C05454=1045.852,-21.922,423.875,169.880,34.118,156.433
C05455=1045.858,-21.672,423.861,169.882,34.118,156.433
C05456=1045.864,-21.423,423.847,169.883,34.120,156.434
C05457=1045.870,-21.174,423.834,169.885,34.121,156.434
C05458=1045.877,-20.923,423.819,169.887,34.122,156.434
C05459=1045.883,-20.675,423.805,169.889,34.124,156.434
C05460=1045.890,-20.425,423.792,169.891,34.125,156.434
C05461=1045.895,-20.175,423.778,169.893,34.126,156.434
C05462=1045.902,-19.925,423.764,169.895,34.127,156.435
C05463=1045.908,-19.676,423.750,169.897,34.129,156.435
C05464=1045.916,-19.394,423.734,169.899,34.130,156.435
C05465=1045.922,-19.113,423.719,169.901,34.131,156.435
C05466=1045.930,-18.831,423.702,169.904,34.133,156.435
C05467=1045.937,-18.550,423.687,169.906,34.134,156.436
C05468=1045.943,-18.300,423.673,169.908,34.136,156.436
C05469=1045.949,-18.051,423.658,169.910,34.137,156.436
C05470=1045.956,-17.801,423.645,169.912,34.138,156.436
C05471=1045.962,-17.552,423.632,169.914,34.140,156.436
C05472=1045.969,-17.302,423.617,169.915,34.141,156.436
C05473=1045.975,-17.053,423.603,169.917,34.142,156.437
C05474=1045.981,-16.803,423.588,169.919,34.143,156.437
C05475=1045.987,-16.554,423.575,169.921,34.145,156.437
C05476=1045.993,-16.303,423.561,169.923,34.146,156.437
C05477=1046.001,-16.054,423.547,169.925,34.147,156.437
C05478=1046.007,-15.805,423.533,169.927,34.148,156.438
C05479=1046.013,-15.555,423.518,169.929,34.150,156.438
C05480=1046.019,-15.306,423.505,169.931,34.151,156.438
C05481=1046.026,-15.056,423.490,169.933,34.152,156.438
C05482=1046.031,-14.807,423.476,169.935,34.154,156.438
C05483=1046.038,-14.557,423.462,169.938,34.155,156.439
C05484=1046.044,-14.308,423.448,169.940,34.157,156.439
C05485=1046.050,-14.058,423.433,169.941,34.158,156.439
C05486=1046.057,-13.808,423.419,169.943,34.159,156.439
C05487=1046.063,-13.559,423.405,169.945,34.161,156.439
C05488=1046.069,-13.309,423.391,169.947,34.162,156.440
C05489=1046.075,-13.060,423.377,169.949,34.163,156.440
C05490=1046.082,-12.810,423.362,169.951,34.165,156.440
C05491=1046.087,-12.561,423.348,169.953,34.166,156.440
C05492=1046.094,-12.312,423.333,169.955,34.168,156.440
C05493=1046.100,-12.062,423.320,169.957,34.169,156.441
C05494=1046.106,-11.812,423.305,169.958,34.170,156.441
C05495=1046.113,-11.562,423.291,169.960,34.172,156.441
C05496=1046.119,-11.314,423.276,169.962,34.173,156.441
C05497=1046.125,-11.064,423.262,169.964,34.174,156.441
C05498=1046.131,-10.815,423.248,169.966,34.176,156.442
C05499=1046.138,-10.565,423.233,169.968,34.177,156.442
C05500=1046.144,-10.315,423.218,169.970,34.178,156.442
C05501=1046.150,-10.066,423.205,169.972,34.180,156.442
C05502=1046.157,-9.816,423.190,169.974,34.181,156.442
C05503=1046.163,-9.567,423.175,169.975,34.183,156.443
C05504=1046.169,-9.317,423.161,169.977,34.184,156.443
C05505=1046.176,-9.068,423.147,169.979,34.185,156.443
C05506=1046.182,-8.818,423.132,169.981,34.187,156.443
C05507=1046.188,-8.569,423.118,169.983,34.188,156.443
C05508=1046.195,-8.319,423.104,169.985,34.189,156.444
C05509=1046.201,-8.070,423.089,169.987,34.191,156.444
C05510=1046.207,-7.821,423.074,169.989,34.192,156.444
C05511=1046.213,-7.570,423.060,169.990,34.194,156.444
C05512=1046.220,-7.321,423.046,169.992,34.195,156.444
C05513=1046.226,-7.072,423.031,169.994,34.196,156.445
C05514=1046.232,-6.822,423.016,169.996,34.198,156.445
C05515=1046.239,-6.572,423.003,169.998,34.199,156.445
C05516=1046.245,-6.323,422.988,170.001,34.200,156.445
C05517=1046.251,-6.074,422.973,170.003,34.202,156.445
C05518=1046.258,-5.824,422.958,170.005,34.203,156.446
C05519=1046.264,-5.575,422.945,170.006,34.205,156.446
C05520=1046.270,-5.325,422.930,170.008,34.206,156.446
C05521=1046.277,-5.076,422.915,170.010,34.207,156.446
C05522=1046.283,-4.826,422.900,170.012,34.209,156.446
C05523=1046.290,-4.577,422.886,170.014,34.210,156.447
C05524=1046.296,-4.328,422.871,170.016,34.211,156.447
C05525=1046.302,-4.077,422.857,170.018,34.213,156.447
C05526=1046.308,-3.828,422.842,170.019,34.214,156.447
C05527=1046.315,-3.579,422.828,170.021,34.215,156.447
C05528=1046.322,-3.296,422.811,170.023,34.217,156.448
C05529=1046.329,-3.012,422.794,170.025,34.219,156.448
C05530=1046.336,-2.729,422.778,170.028,34.220,156.448
C05531=1046.343,-2.446,422.760,170.030,34.222,156.448
C05532=1046.350,-2.196,422.745,170.031,34.224,156.449
C05533=1046.355,-1.947,422.731,170.033,34.225,156.449
C05534=1046.362,-1.698,422.716,170.035,34.226,156.449
C05535=1046.368,-1.448,422.701,170.037,34.228,156.449
C05536=1046.374,-1.199,422.686,170.039,34.230,156.450
C05537=1046.380,-0.950,422.671,170.041,34.231,156.450
C05538=1046.387,-0.700,422.657,170.042,34.232,156.450
C05539=1046.393,-0.450,422.642,170.044,34.234,156.450
C05540=1046.399,-0.201,422.627,170.046,34.236,156.450
C05541=1046.404,0.049,422.611,170.048,34.237,156.451
C05542=1046.411,0.298,422.597,170.050,34.239,156.451
C05543=1046.417,0.548,422.582,170.052,34.240,156.451
C05544=1046.423,0.797,422.567,170.054,34.241,156.451
C05545=1046.429,1.047,422.552,170.056,34.243,156.452
C05546=1046.436,1.296,422.537,170.058,34.245,156.452
C05547=1046.442,1.546,422.522,170.060,34.246,156.452
C05548=1046.448,1.795,422.508,170.062,34.247,156.452
C05549=1046.454,2.045,422.493,170.063,34.249,156.452
C05550=1046.461,2.294,422.478,170.065,34.250,156.453
C05551=1046.467,2.544,422.463,170.067,34.252,156.453
C05552=1046.474,2.793,422.447,170.069,34.253,156.453
C05553=1046.480,3.042,422.433,170.071,34.255,156.453
C05554=1046.486,3.292,422.418,170.072,34.256,156.454
C05555=1046.492,3.541,422.403,170.074,34.257,156.454
C05556=1046.498,3.791,422.387,170.076,34.259,156.454
C05557=1046.504,4.041,422.372,170.078,34.261,156.454
C05558=1046.511,4.290,422.357,170.080,34.262,156.454
C05559=1046.517,4.539,422.342,170.081,34.264,156.455
C05560=1046.523,4.788,422.327,170.083,34.265,156.455
C05561=1046.530,5.038,422.312,170.085,34.267,156.455
C05562=1046.536,5.288,422.297,170.087,34.268,156.455
C05563=1046.542,5.537,422.282,170.089,34.270,156.456
C05564=1046.549,5.787,422.267,170.090,34.271,156.456
C05565=1046.555,6.035,422.252,170.092,34.272,156.456
C05566=1046.561,6.285,422.237,170.094,34.274,156.456
C05567=1046.567,6.535,422.221,170.097,34.276,156.457
C05568=1046.573,6.785,422.206,170.099,34.277,156.457
C05569=1046.580,7.034,422.191,170.100,34.278,156.457
C05570=1046.586,7.283,422.176,170.102,34.280,156.457
C05571=1046.593,7.533,422.161,170.104,34.282,156.457
C05572=1046.599,7.783,422.146,170.106,34.283,156.458
C05573=1046.606,8.032,422.130,170.108,34.284,156.458
C05574=1046.612,8.281,422.116,170.109,34.286,156.458
C05575=1046.617,8.531,422.100,170.111,34.287,156.458
C05576=1046.624,8.780,422.085,170.113,34.289,156.459
C05577=1046.630,9.029,422.070,170.115,34.291,156.459
C05578=1046.637,9.279,422.055,170.117,34.292,156.459
C05579=1046.643,9.529,422.040,170.118,34.293,156.459
C05580=1046.650,9.778,422.024,170.120,34.295,156.459
C05581=1046.656,10.027,422.009,170.122,34.297,156.460
C05582=1046.662,10.277,421.994,170.124,34.298,156.460
C05583=1046.668,10.526,421.978,170.126,34.299,156.460
C05584=1046.675,10.776,421.963,170.127,34.301,156.460
C05585=1046.681,11.026,421.948,170.129,34.302,156.461
C05586=1046.688,11.275,421.932,170.131,34.304,156.461
C05587=1046.694,11.524,421.917,170.133,34.305,156.461
C05588=1046.701,11.774,421.902,170.135,34.307,156.461
C05589=1046.707,12.023,421.887,170.136,34.308,156.461
C05590=1046.713,12.273,421.871,170.139,34.309,156.462
C05591=1046.720,12.522,421.856,170.141,34.311,156.462
C05592=1046.727,12.807,421.838,170.143,34.313,156.462
C05593=1046.734,13.092,421.821,170.145,34.315,156.463
C05594=1046.741,13.378,421.804,170.147,34.316,156.463
C05595=1046.749,13.663,421.786,170.149,34.318,156.463
C05596=1046.756,13.912,421.770,170.151,34.319,156.463
C05597=1046.762,14.162,421.755,170.153,34.321,156.463
C05598=1046.768,14.411,421.739,170.154,34.322,156.464
C05599=1046.774,14.661,421.724,170.156,34.324,156.464
C05600=1046.781,14.910,421.708,170.158,34.325,156.464
C05601=1046.787,15.160,421.693,170.160,34.327,156.464
C05602=1046.793,15.409,421.677,170.161,34.329,156.465
C05603=1046.799,15.659,421.662,170.163,34.330,156.465
C05604=1046.806,15.908,421.646,170.165,34.332,156.465
C05605=1046.812,16.157,421.631,170.167,34.333,156.465
C05606=1046.818,16.407,421.615,170.168,34.335,156.466
C05607=1046.825,16.656,421.599,170.170,34.336,156.466
C05608=1046.830,16.906,421.584,170.172,34.338,156.466
C05609=1046.837,17.155,421.568,170.174,34.340,156.466
C05610=1046.843,17.404,421.553,170.175,34.341,156.467
C05611=1046.849,17.654,421.537,170.178,34.343,156.467
C05612=1046.856,17.903,421.522,170.180,34.344,156.467
C05613=1046.862,18.153,421.506,170.182,34.346,156.467
C05614=1046.868,18.402,421.490,170.183,34.347,156.468
C05615=1046.875,18.651,421.475,170.185,34.349,156.468
C05616=1046.881,18.901,421.459,170.187,34.350,156.468
C05617=1046.887,19.150,421.443,170.189,34.352,156.468
C05618=1046.893,19.400,421.427,170.190,34.353,156.469
C05619=1046.900,19.649,421.412,170.192,34.355,156.469
C05620=1046.906,19.898,421.396,170.194,34.357,156.469
C05621=1046.912,20.148,421.381,170.196,34.358,156.469
C05622=1046.918,20.397,421.364,170.197,34.360,156.470
C05623=1046.925,20.646,421.349,170.199,34.362,156.470
C05624=1046.930,20.896,421.333,170.201,34.363,156.470
C05625=1046.937,21.145,421.317,170.203,34.365,156.470
C05626=1046.943,21.394,421.301,170.204,34.366,156.471
C05627=1046.950,21.644,421.285,170.206,34.368,156.471
C05628=1046.956,21.894,421.270,170.208,34.370,156.471
C05629=1046.963,22.143,421.254,170.209,34.371,156.471
C05630=1046.969,22.393,421.238,170.212,34.373,156.472
C05631=1046.975,22.642,421.222,170.214,34.374,156.472
C05632=1046.981,22.892,421.207,170.216,34.376,156.472
C05633=1046.987,23.141,421.190,170.217,34.377,156.472
C05634=1046.994,23.390,421.175,170.219,34.379,156.473
C05635=1046.999,23.639,421.158,170.221,34.381,156.473
C05636=1047.006,23.888,421.143,170.223,34.382,156.473
C05637=1047.012,24.139,421.127,170.224,34.383,156.473
C05638=1047.019,24.388,421.111,170.226,34.385,156.474
C05639=1047.025,24.637,421.095,170.228,34.387,156.474
C05640=1047.031,24.887,421.079,170.229,34.388,156.474
C05641=1047.038,25.136,421.063,170.231,34.390,156.474
C05642=1047.044,25.385,421.047,170.233,34.391,156.475
C05643=1047.050,25.635,421.032,170.235,34.393,156.475
C05644=1047.057,25.885,421.015,170.236,34.395,156.475
C05645=1047.063,26.134,420.999,170.238,34.396,156.475
C05646=1047.069,26.383,420.983,170.240,34.398,156.476
C05647=1047.075,26.633,420.967,170.241,34.399,156.476
C05648=1047.082,26.882,420.951,170.244,34.401,156.476
C05649=1047.088,27.131,420.935,170.246,34.403,156.476
C05650=1047.094,27.381,420.918,170.248,34.404,156.477
C05651=1047.101,27.630,420.903,170.249,34.406,156.477
C05652=1047.107,27.879,420.887,170.251,34.407,156.477
C05653=1047.113,28.129,420.870,170.253,34.409,156.477
C05654=1047.119,28.378,420.855,170.254,34.411,156.478
C05655=1047.125,28.628,420.839,170.256,34.413,156.478
C05656=1047.133,28.914,420.820,170.258,34.414,156.478
C05657=1047.140,29.200,420.802,170.260,34.416,156.479
C05658=1047.147,29.486,420.783,170.262,34.418,156.479
C05659=1047.154,29.773,420.764,170.264,34.420,156.479
C05660=1047.160,30.022,420.748,170.266,34.421,156.479
C05661=1047.167,30.271,420.732,170.267,34.423,156.480
C05662=1047.173,30.521,420.715,170.269,34.425,156.480
C05663=1047.179,30.771,420.699,170.271,34.427,156.480
C05664=1047.185,31.020,420.683,170.272,34.428,156.480
C05665=1047.191,31.270,420.667,170.275,34.430,156.481
C05666=1047.198,31.519,420.651,170.277,34.431,156.481
C05667=1047.204,31.769,420.634,170.279,34.433,156.481
C05668=1047.210,32.018,420.618,170.280,34.434,156.481
C05669=1047.216,32.267,420.602,170.282,34.436,156.482
C05670=1047.222,32.517,420.586,170.284,34.438,156.482
C05671=1047.230,32.766,420.569,170.285,34.440,156.482
C05672=1047.236,33.015,420.553,170.287,34.441,156.483
C05673=1047.242,33.264,420.536,170.289,34.443,156.483
C05674=1047.248,33.514,420.520,170.290,34.444,156.483
C05675=1047.254,33.764,420.503,170.292,34.446,156.483
C05676=1047.261,34.013,420.488,170.294,34.448,156.484
C05677=1047.267,34.262,420.471,170.295,34.450,156.484
C05678=1047.273,34.512,420.455,170.297,34.451,156.484
C05679=1047.280,34.761,420.438,170.299,34.453,156.484
C05680=1047.286,35.010,420.422,170.301,34.454,156.485
C05681=1047.292,35.260,420.405,170.303,34.456,156.485
C05682=1047.298,35.509,420.390,170.305,34.458,156.485
C05683=1047.305,35.759,420.373,170.307,34.460,156.486
C05684=1047.311,36.008,420.356,170.308,34.461,156.486
C05685=1047.317,36.257,420.340,170.310,34.462,156.486
C05686=1047.324,36.507,420.323,170.312,34.464,156.486
C05687=1047.330,36.756,420.307,170.313,34.465,156.487
C05688=1047.336,37.006,420.291,170.315,34.467,156.487
C05689=1047.343,37.255,420.274,170.317,34.469,156.487
C05690=1047.349,37.504,420.258,170.318,34.471,156.487
C05691=1047.355,37.753,420.241,170.320,34.472,156.488
C05692=1047.362,38.003,420.224,170.322,34.474,156.488
C05693=1047.368,38.252,420.208,170.323,34.476,156.488
C05694=1047.374,38.502,420.192,170.325,34.477,156.488
C05695=1047.380,38.751,420.175,170.327,34.479,156.489
C05696=1047.387,39.000,420.158,170.328,34.481,156.489
C05697=1047.393,39.250,420.142,170.331,34.483,156.489
C05698=1047.398,39.499,420.124,170.333,34.484,156.490
C05699=1047.405,39.749,420.108,170.334,34.486,156.490
C05700=1047.411,39.998,420.091,170.336,34.488,156.490
C05701=1047.417,40.247,420.074,170.338,34.489,156.490
C05702=1047.423,40.497,420.058,170.339,34.491,156.491
C05703=1047.429,40.746,420.041,170.341,34.492,156.491
C05704=1047.436,40.995,420.024,170.343,34.494,156.491
C05705=1047.442,41.245,420.008,170.344,34.496,156.491
C05706=1047.448,41.494,419.991,170.346,34.498,156.492
C05707=1047.454,41.743,419.975,170.348,34.500,156.492
C05708=1047.461,41.993,419.958,170.349,34.501,156.492
C05709=1047.467,42.242,419.941,170.351,34.503,156.493
C05710=1047.473,42.491,419.925,170.353,34.504,156.493
C05711=1047.480,42.741,419.907,170.355,34.506,156.493
C05712=1047.486,42.990,419.891,170.357,34.508,156.493
C05713=1047.491,43.239,419.874,170.359,34.510,156.494
C05714=1047.498,43.489,419.857,170.360,34.511,156.494
C05715=1047.504,43.738,419.840,170.362,34.513,156.494
C05716=1047.511,43.988,419.823,170.364,34.515,156.495
C05717=1047.516,44.237,419.806,170.365,34.517,156.495
C05718=1047.522,44.486,419.790,170.367,34.518,156.495
C05719=1047.529,44.736,419.772,170.369,34.520,156.495
C05720=1047.536,45.022,419.753,170.371,34.522,156.496
C05721=1047.543,45.308,419.733,170.372,34.524,156.496
C05722=1047.549,45.595,419.714,170.374,34.526,156.496
C05723=1047.557,45.881,419.695,170.376,34.528,156.497
C05724=1047.562,46.130,419.678,170.378,34.530,156.497
C05725=1047.569,46.380,419.660,170.380,34.532,156.497
C05726=1047.575,46.629,419.644,170.382,34.533,156.498
C05727=1047.581,46.879,419.626,170.384,34.535,156.498
C05728=1047.587,47.128,419.610,170.385,34.537,156.498
C05729=1047.593,47.377,419.593,170.387,34.538,156.498
C05730=1047.600,47.626,419.575,170.389,34.540,156.499
C05731=1047.606,47.876,419.559,170.390,34.542,156.499
C05732=1047.612,48.125,419.541,170.392,34.544,156.499
C05733=1047.618,48.374,419.524,170.394,34.545,156.500
C05734=1047.624,48.624,419.507,170.395,34.547,156.500
C05735=1047.631,48.873,419.490,170.397,34.549,156.500
C05736=1047.636,49.122,419.473,170.398,34.551,156.501
C05737=1047.643,49.372,419.456,170.400,34.553,156.501
C05738=1047.649,49.621,419.439,170.402,34.554,156.501
C05739=1047.655,49.871,419.421,170.404,34.556,156.501
C05740=1047.661,50.120,419.405,170.406,34.558,156.502
C05741=1047.667,50.369,419.388,170.408,34.559,156.502
C05742=1047.673,50.618,419.370,170.409,34.561,156.502
C05743=1047.679,50.868,419.354,170.411,34.563,156.503
C05744=1047.686,51.117,419.336,170.413,34.564,156.503
C05745=1047.692,51.366,419.319,170.414,34.566,156.503
C05746=1047.699,51.616,419.301,170.416,34.568,156.503
C05747=1047.704,51.865,419.285,170.418,34.570,156.504
C05748=1047.711,52.115,419.267,170.419,34.572,156.504
C05749=1047.717,52.363,419.250,170.421,34.574,156.504
C05750=1047.723,52.613,419.232,170.422,34.575,156.505
C05751=1047.729,52.862,419.215,170.424,34.577,156.505
C05752=1047.736,53.112,419.199,170.427,34.579,156.505
C05753=1047.741,53.361,419.181,170.428,34.580,156.505
C05754=1047.748,53.610,419.164,170.430,34.582,156.506
C05755=1047.754,53.859,419.146,170.432,34.583,156.506
C05756=1047.761,54.109,419.129,170.433,34.585,156.506
C05757=1047.767,54.358,419.113,170.435,34.587,156.507
C05758=1047.773,54.608,419.095,170.437,34.589,156.507
C05759=1047.779,54.857,419.078,170.438,34.590,156.507
C05760=1047.786,55.106,419.060,170.440,34.592,156.507
C05761=1047.792,55.356,419.042,170.442,34.594,156.508
C05762=1047.798,55.605,419.025,170.443,34.596,156.508
C05763=1047.804,55.854,419.008,170.445,34.598,156.508
C05764=1047.810,56.104,418.991,170.446,34.599,156.509
C05765=1047.817,56.353,418.974,170.449,34.601,156.509
C05766=1047.823,56.602,418.956,170.451,34.602,156.509
C05767=1047.830,56.852,418.939,170.452,34.604,156.509
C05768=1047.835,57.101,418.921,170.454,34.606,156.510
C05769=1047.842,57.350,418.904,170.456,34.607,156.510
C05770=1047.849,57.600,418.887,170.457,34.609,156.510
C05771=1047.854,57.849,418.869,170.459,34.611,156.511
C05772=1047.861,58.098,418.852,170.461,34.613,156.511
C05773=1047.867,58.347,418.834,170.462,34.615,156.511
C05774=1047.874,58.596,418.817,170.464,34.616,156.511
C05775=1047.880,58.846,418.800,170.466,34.618,156.512
C05776=1047.886,59.095,418.782,170.467,34.620,156.512
C05777=1047.893,59.344,418.765,170.469,34.621,156.512
C05778=1047.899,59.595,418.748,170.472,34.623,156.513
C05779=1047.905,59.843,418.731,170.473,34.624,156.513
C05780=1047.911,60.093,418.713,170.475,34.626,156.513
C05781=1047.917,60.342,418.696,170.476,34.628,156.513
C05782=1047.924,60.591,418.678,170.478,34.630,156.514
C05783=1047.931,60.840,418.660,170.480,34.632,156.514
C05784=1047.937,61.126,418.640,170.482,34.634,156.514
C05785=1047.944,61.412,418.620,170.484,34.635,156.515
C05786=1047.953,61.699,418.600,170.485,34.637,156.515
C05787=1047.960,61.985,418.580,170.487,34.639,156.515
C05788=1047.966,62.234,418.562,170.489,34.641,156.516
C05789=1047.972,62.483,418.545,170.491,34.643,156.516
C05790=1047.978,62.733,418.527,170.493,34.645,156.516
C05791=1047.985,62.982,418.510,170.495,34.646,156.516
C05792=1047.991,63.231,418.492,170.497,34.648,156.517
C05793=1047.998,63.480,418.474,170.498,34.649,156.517
C05794=1048.005,63.730,418.457,170.500,34.651,156.517
C05795=1048.010,63.979,418.439,170.502,34.652,156.517
C05796=1048.016,64.228,418.421,170.503,34.654,156.518
C05797=1048.023,64.478,418.404,170.505,34.656,156.518
C05798=1048.029,64.727,418.386,170.506,34.658,156.518
C05799=1048.035,64.977,418.369,170.508,34.660,156.519
C05800=1048.042,65.225,418.351,170.510,34.661,156.519
C05801=1048.048,65.475,418.333,170.511,34.663,156.519
C05802=1048.054,65.724,418.315,170.513,34.665,156.520
C05803=1048.060,65.974,418.298,170.516,34.667,156.520
C05804=1048.067,66.223,418.280,170.517,34.669,156.520
C05805=1048.072,66.472,418.262,170.519,34.671,156.521
C05806=1048.079,66.721,418.244,170.520,34.672,156.521
C05807=1048.085,66.971,418.226,170.522,34.674,156.521
C05808=1048.091,67.220,418.209,170.524,34.676,156.521
C05809=1048.097,67.469,418.190,170.525,34.677,156.522
C05810=1048.104,67.718,418.173,170.527,34.679,156.522
C05811=1048.110,67.967,418.155,170.529,34.681,156.522
C05812=1048.116,68.217,418.136,170.530,34.683,156.523
C05813=1048.122,68.466,418.119,170.532,34.684,156.523
C05814=1048.129,68.716,418.101,170.533,34.686,156.523
C05815=1048.135,68.964,418.083,170.536,34.688,156.524
C05816=1048.141,69.214,418.065,170.538,34.690,156.524
C05817=1048.147,69.464,418.047,170.539,34.691,156.524
C05818=1048.154,69.713,418.028,170.541,34.693,156.524
C05819=1048.160,69.962,418.011,170.543,34.695,156.525
C05820=1048.166,70.211,417.994,170.544,34.697,156.525
C05821=1048.172,70.460,417.975,170.546,34.698,156.525
C05822=1048.178,70.709,417.957,170.547,34.700,156.526
C05823=1048.184,70.959,417.939,170.549,34.702,156.526
C05824=1048.190,71.208,417.921,170.551,34.704,156.526
C05825=1048.197,71.458,417.903,170.552,34.705,156.527
C05826=1048.202,71.706,417.884,170.555,34.707,156.527
C05827=1048.208,71.956,417.867,170.557,34.709,156.527
C05828=1048.215,72.206,417.849,170.558,34.711,156.528
C05829=1048.222,72.455,417.831,170.560,34.713,156.528
C05830=1048.227,72.704,417.813,170.561,34.715,156.528
C05831=1048.234,72.953,417.794,170.563,34.716,156.528
C05832=1048.240,73.203,417.776,170.565,34.718,156.529
C05833=1048.246,73.452,417.758,170.566,34.720,156.529
C05834=1048.252,73.701,417.740,170.568,34.722,156.529
C05835=1048.258,73.950,417.722,170.570,34.724,156.530
C05836=1048.264,74.200,417.704,170.571,34.726,156.530
C05837=1048.271,74.449,417.685,170.574,34.727,156.530
C05838=1048.277,74.699,417.667,170.575,34.729,156.530
C05839=1048.283,74.947,417.649,170.577,34.731,156.531
C05840=1048.289,75.197,417.631,170.579,34.733,156.531
C05841=1048.295,75.446,417.612,170.580,34.735,156.531
C05842=1048.302,75.695,417.595,170.582,34.736,156.532
C05843=1048.309,75.944,417.576,170.584,34.738,156.532
C05844=1048.314,76.193,417.559,170.585,34.740,156.532
C05845=1048.320,76.443,417.540,170.587,34.742,156.533
C05846=1048.327,76.692,417.521,170.588,34.744,156.533
C05847=1048.333,76.941,417.503,170.590,34.745,156.533
C05848=1048.340,77.227,417.482,170.592,34.747,156.534
C05849=1048.347,77.513,417.461,170.595,34.749,156.534
C05850=1048.354,77.799,417.440,170.597,34.751,156.534
C05851=1048.361,78.084,417.419,170.598,34.753,156.535
C05852=1048.367,78.334,417.401,170.600,34.755,156.535
C05853=1048.374,78.583,417.383,170.602,34.757,156.535
C05854=1048.380,78.832,417.364,170.603,34.758,156.536
C05855=1048.386,79.082,417.345,170.605,34.760,156.536
C05856=1048.392,79.331,417.327,170.607,34.762,156.536
C05857=1048.398,79.580,417.308,170.608,34.764,156.537
C05858=1048.404,79.829,417.291,170.610,34.766,156.537
C05859=1048.410,80.078,417.272,170.612,34.768,156.537
C05860=1048.416,80.328,417.253,170.614,34.770,156.538
C05861=1048.422,80.577,417.234,170.616,34.772,156.538
C05862=1048.429,80.827,417.216,170.617,34.773,156.538
C05863=1048.434,81.075,417.198,170.619,34.775,156.538
C05864=1048.441,81.324,417.179,170.620,34.777,156.539
C05865=1048.447,81.574,417.160,170.622,34.779,156.539
C05866=1048.453,81.823,417.142,170.624,34.781,156.539
C05867=1048.459,82.073,417.123,170.625,34.783,156.540
C05868=1048.466,82.322,417.105,170.627,34.784,156.540
C05869=1048.472,82.571,417.086,170.630,34.786,156.540
C05870=1048.477,82.821,417.068,170.631,34.788,156.541
C05871=1048.483,83.069,417.049,170.633,34.790,156.541
C05872=1048.490,83.318,417.031,170.634,34.792,156.541
C05873=1048.496,83.568,417.012,170.636,34.794,156.542
C05874=1048.502,83.817,416.993,170.638,34.796,156.542
C05875=1048.508,84.066,416.974,170.639,34.797,156.542
C05876=1048.514,84.316,416.956,170.641,34.799,156.543
C05877=1048.521,84.565,416.937,170.643,34.801,156.543
C05878=1048.527,84.814,416.919,170.644,34.803,156.543
C05879=1048.533,85.064,416.900,170.647,34.805,156.544
C05880=1048.539,85.313,416.881,170.648,34.806,156.544
C05881=1048.546,85.562,416.862,170.650,34.808,156.544
C05882=1048.552,85.811,416.844,170.652,34.810,156.544
C05883=1048.558,86.060,416.824,170.653,34.812,156.545
C05884=1048.563,86.309,416.807,170.655,34.814,156.545
C05885=1048.570,86.558,416.788,170.657,34.816,156.545
C05886=1048.576,86.808,416.770,170.658,34.817,156.546
C05887=1048.583,87.057,416.751,170.660,34.819,156.546
C05888=1048.588,87.306,416.732,170.661,34.821,156.546
C05889=1048.595,87.555,416.713,170.663,34.823,156.547
C05890=1048.601,87.804,416.694,170.666,34.825,156.547
C05891=1048.608,88.053,416.676,170.667,34.826,156.547
C05892=1048.613,88.303,416.656,170.669,34.828,156.548
C05893=1048.620,88.552,416.638,170.671,34.830,156.548
C05894=1048.626,88.801,416.619,170.672,34.832,156.548
C05895=1048.632,89.050,416.600,170.674,34.834,156.549
C05896=1048.638,89.300,416.581,170.676,34.835,156.549
C05897=1048.645,89.549,416.563,170.677,34.837,156.549
C05898=1048.651,89.798,416.544,170.679,34.839,156.549
C05899=1048.657,90.047,416.525,170.680,34.841,156.550
C05900=1048.663,90.297,416.506,170.683,34.843,156.550
C05901=1048.670,90.546,416.487,170.685,34.844,156.550
C05902=1048.675,90.795,416.468,170.686,34.846,156.551
C05903=1048.682,91.044,416.450,170.688,34.848,156.551
C05904=1048.687,91.294,416.430,170.690,34.850,156.551
C05905=1048.694,91.543,416.412,170.691,34.852,156.552
C05906=1048.699,91.792,416.392,170.693,34.854,156.552
C05907=1048.706,92.041,416.373,170.694,34.855,156.552
C05908=1048.712,92.290,416.354,170.696,34.857,156.553
C05909=1048.718,92.539,416.335,170.698,34.859,156.553
C05910=1048.724,92.789,416.316,170.700,34.861,156.553
C05911=1048.730,93.038,416.297,170.702,34.863,156.554
C05912=1048.738,93.323,416.275,170.704,34.865,156.554
C05913=1048.745,93.610,416.253,170.706,34.867,156.554
C05914=1048.751,93.895,416.231,170.708,34.870,156.555
C05915=1048.758,94.181,416.209,170.709,34.871,156.555
C05916=1048.765,94.431,416.190,170.711,34.873,156.555
C05917=1048.770,94.680,416.171,170.713,34.875,156.556
C05918=1048.777,94.929,416.152,170.714,34.877,156.556
C05919=1048.783,95.178,416.133,170.717,34.879,156.556
C05920=1048.789,95.427,416.114,170.719,34.881,156.557
C05921=1048.795,95.677,416.095,170.720,34.882,156.557
C05922=1048.802,95.925,416.075,170.722,34.884,156.557
C05923=1048.807,96.174,416.056,170.724,34.886,156.558
C05924=1048.814,96.424,416.037,170.725,34.888,156.558
C05925=1048.819,96.673,416.018,170.727,34.890,156.558
C05926=1048.825,96.922,415.998,170.728,34.892,156.559
C05927=1048.832,97.172,415.979,170.730,34.894,156.559
C05928=1048.838,97.421,415.960,170.733,34.896,156.559
C05929=1048.845,97.670,415.941,170.734,34.897,156.560
C05930=1048.851,97.919,415.921,170.736,34.899,156.560
C05931=1048.857,98.168,415.903,170.738,34.901,156.560
C05932=1048.863,98.418,415.883,170.739,34.903,156.561
C05933=1048.869,98.666,415.864,170.741,34.905,156.561
C05934=1048.875,98.915,415.845,170.743,34.907,156.561
C05935=1048.881,99.165,415.826,170.744,34.909,156.562
C05936=1048.888,99.414,415.806,170.746,34.911,156.562
C05937=1048.894,99.664,415.787,170.748,34.912,156.562
C05938=1048.901,99.912,415.767,170.750,34.914,156.563
C05939=1048.906,100.161,415.748,170.752,34.916,156.563
C05940=1048.913,100.411,415.729,170.754,34.918,156.563
C05941=1048.919,100.659,415.709,170.755,34.920,156.564
C05942=1048.924,100.909,415.690,170.757,34.921,156.564
C05943=1048.931,101.159,415.671,170.759,34.923,156.564
C05944=1048.937,101.407,415.651,170.760,34.925,156.565
C05945=1048.943,101.657,415.632,170.762,34.927,156.565
C05946=1048.949,101.906,415.612,170.763,34.929,156.565
C05947=1048.955,102.155,415.593,170.766,34.931,156.566
C05948=1048.961,102.404,415.573,170.768,34.933,156.566
C05949=1048.967,102.653,415.554,170.769,34.935,156.566
C05950=1048.973,102.902,415.534,170.771,34.937,156.567
C05951=1048.979,103.152,415.515,170.773,34.939,156.567
C05952=1048.985,103.401,415.495,170.774,34.941,156.567
C05953=1048.991,103.650,415.475,170.776,34.942,156.568
C05954=1048.997,103.899,415.455,170.778,34.944,156.568
C05955=1049.004,104.148,415.437,170.779,34.946,156.568
C05956=1049.010,104.397,415.417,170.782,34.948,156.569
C05957=1049.016,104.647,415.396,170.784,34.950,156.569
C05958=1049.022,104.896,415.377,170.785,34.952,156.569
C05959=1049.028,105.145,415.357,170.787,34.953,156.569
C05960=1049.033,105.394,415.338,170.788,34.955,156.570
C05961=1049.040,105.643,415.319,170.790,34.957,156.570
C05962=1049.046,105.892,415.299,170.792,34.959,156.571
C05963=1049.052,106.142,415.279,170.793,34.961,156.571
C05964=1049.058,106.391,415.259,170.795,34.963,156.571
C05965=1049.064,106.640,415.240,170.798,34.965,156.572
C05966=1049.070,106.889,415.220,170.799,34.967,156.572
C05967=1049.077,107.139,415.201,170.801,34.969,156.572
C05968=1049.083,107.387,415.181,170.803,34.971,156.573
C05969=1049.089,107.636,415.161,170.804,34.972,156.573
C05970=1049.095,107.886,415.142,170.806,34.974,156.573
C05971=1049.101,108.134,415.122,170.808,34.976,156.574
C05972=1049.107,108.384,415.101,170.809,34.978,156.574
C05973=1049.114,108.633,415.083,170.811,34.980,156.574
C05974=1049.120,108.882,415.063,170.814,34.982,156.575
C05975=1049.126,109.131,415.043,170.815,34.984,156.575
C05976=1049.133,109.417,415.020,170.817,34.986,156.575
C05977=1049.140,109.702,414.998,170.819,34.988,156.576
C05978=1049.147,109.988,414.975,170.821,34.990,156.576
C05979=1049.154,110.274,414.952,170.823,34.992,156.576
C05980=1049.161,110.524,414.932,170.825,34.994,156.577
C05981=1049.167,110.772,414.912,170.826,34.996,156.577
C05982=1049.172,111.022,414.893,170.829,34.998,156.577
C05983=1049.178,111.271,414.873,170.831,35.000,156.578
C05984=1049.185,111.520,414.853,170.833,35.002,156.578
C05985=1049.191,111.769,414.833,170.834,35.004,156.578
C05986=1049.197,112.018,414.813,170.836,35.006,156.579
C05987=1049.203,112.268,414.793,170.838,35.008,156.579
C05988=1049.209,112.517,414.773,170.839,35.009,156.579
C05989=1049.215,112.766,414.753,170.841,35.011,156.580
C05990=1049.221,113.014,414.733,170.843,35.013,156.580
C05991=1049.228,113.264,414.713,170.845,35.015,156.580
C05992=1049.234,113.513,414.693,170.847,35.017,156.581
C05993=1049.240,113.762,414.674,170.849,35.019,156.581
C05994=1049.246,114.012,414.653,170.850,35.021,156.581
C05995=1049.251,114.261,414.633,170.852,35.023,156.582
C05996=1049.257,114.510,414.613,170.854,35.025,156.582
C05997=1049.263,114.758,414.593,170.855,35.027,156.582
C05998=1049.270,115.008,414.572,170.857,35.028,156.583
C05999=1049.275,115.257,414.552,170.860,35.031,156.583
C06000=1049.281,115.506,414.532,170.861,35.033,156.584
C06001=1049.287,115.755,414.512,170.863,35.035,156.584
C06002=1049.294,116.004,414.492,170.865,35.037,156.584
C06003=1049.299,116.253,414.471,170.866,35.039,156.585
C06004=1049.305,116.502,414.451,170.868,35.041,156.585
C06005=1049.312,116.752,414.431,170.870,35.042,156.585
C06006=1049.318,117.001,414.411,170.871,35.044,156.586
C06007=1049.323,117.250,414.390,170.874,35.046,156.586
C06008=1049.330,117.499,414.370,170.876,35.048,156.586
C06009=1049.336,117.748,414.350,170.877,35.051,156.587
C06010=1049.341,117.997,414.329,170.879,35.053,156.587
C06011=1049.347,118.247,414.309,170.881,35.055,156.587
C06012=1049.353,118.495,414.289,170.882,35.056,156.588
C06013=1049.359,118.744,414.269,170.884,35.058,156.588
C06014=1049.365,118.994,414.248,170.886,35.060,156.588
C06015=1049.371,119.243,414.228,170.888,35.062,156.589
C06016=1049.377,119.491,414.208,170.890,35.064,156.589
C06017=1049.383,119.741,414.187,170.892,35.066,156.590
C06018=1049.389,119.990,414.167,170.893,35.068,156.590
C06019=1049.395,120.238,414.147,170.895,35.070,156.590
C06020=1049.402,120.488,414.127,170.897,35.072,156.591
C06021=1049.407,120.737,414.106,170.899,35.074,156.591
C06022=1049.414,120.987,414.086,170.900,35.076,156.591
C06023=1049.420,121.235,414.066,170.903,35.078,156.592
C06024=1049.425,121.484,414.044,170.905,35.080,156.592
C06025=1049.432,121.733,414.024,170.906,35.082,156.592
C06026=1049.438,121.982,414.004,170.908,35.084,156.593
C06027=1049.444,122.232,413.983,170.910,35.086,156.593
C06028=1049.450,122.481,413.963,170.911,35.087,156.593
C06029=1049.456,122.730,413.943,170.913,35.089,156.594
C06030=1049.462,122.979,413.922,170.915,35.091,156.594
C06031=1049.468,123.228,413.902,170.918,35.093,156.594
C06032=1049.475,123.477,413.881,170.919,35.095,156.595
C06033=1049.480,123.726,413.861,170.921,35.097,156.595
C06034=1049.487,123.975,413.840,170.923,35.099,156.595
C06035=1049.493,124.224,413.820,170.924,35.101,156.596
C06036=1049.499,124.474,413.799,170.926,35.103,156.596
C06037=1049.505,124.723,413.779,170.928,35.105,156.597
C06038=1049.511,124.971,413.758,170.930,35.107,156.597
C06039=1049.517,125.221,413.737,170.932,35.109,156.597
C06040=1049.524,125.506,413.714,170.934,35.111,156.598
C06041=1049.530,125.792,413.691,170.936,35.113,156.598
C06042=1049.537,126.078,413.667,170.938,35.115,156.598
C06043=1049.545,126.364,413.643,170.940,35.118,156.599
C06044=1049.551,126.612,413.623,170.942,35.120,156.599
C06045=1049.558,126.861,413.602,170.944,35.122,156.600
C06046=1049.563,127.111,413.582,170.947,35.124,156.600
C06047=1049.570,127.360,413.561,170.948,35.125,156.600
C06048=1049.576,127.608,413.541,170.950,35.127,156.601
C06049=1049.582,127.858,413.520,170.952,35.129,156.601
C06050=1049.588,128.107,413.500,170.953,35.131,156.601
C06051=1049.594,128.356,413.478,170.955,35.133,156.602
C06052=1049.600,128.605,413.458,170.957,35.135,156.602
C06053=1049.607,128.854,413.437,170.959,35.137,156.602
C06054=1049.612,129.103,413.416,170.961,35.139,156.603
C06055=1049.619,129.352,413.396,170.963,35.141,156.603
C06056=1049.625,129.601,413.375,170.965,35.143,156.603
C06057=1049.631,129.850,413.355,170.967,35.144,156.604
C06058=1049.638,130.099,413.333,170.968,35.146,156.604
C06059=1049.643,130.348,413.313,170.970,35.148,156.604
C06060=1049.650,130.597,413.292,170.972,35.150,156.605
C06061=1049.656,130.846,413.272,170.974,35.152,156.605
C06062=1049.662,131.095,413.250,170.977,35.154,156.605
C06063=1049.669,131.345,413.230,170.978,35.156,156.606
C06064=1049.674,131.593,413.209,170.980,35.158,156.606
C06065=1049.681,131.843,413.188,170.982,35.160,156.606
C06066=1049.686,132.091,413.167,170.984,35.162,156.607
C06067=1049.692,132.341,413.146,170.985,35.164,156.607
C06068=1049.699,132.589,413.126,170.987,35.166,156.607
C06069=1049.705,132.839,413.105,170.990,35.168,156.608
C06070=1049.710,133.088,413.083,170.992,35.170,156.608
C06071=1049.717,133.337,413.063,170.993,35.172,156.609
C06072=1049.723,133.586,413.041,170.995,35.174,156.609
C06073=1049.728,133.835,413.020,170.997,35.176,156.609
C06074=1049.735,134.084,413.000,170.999,35.178,156.610
C06075=1049.741,134.333,412.979,171.000,35.180,156.610
C06076=1049.747,134.582,412.957,171.003,35.182,156.610
C06077=1049.753,134.832,412.937,171.005,35.184,156.611
C06078=1049.759,135.080,412.915,171.007,35.186,156.611
C06079=1049.765,135.329,412.894,171.008,35.188,156.612
C06080=1049.771,135.578,412.874,171.010,35.190,156.612
C06081=1049.777,135.827,412.852,171.012,35.192,156.612
C06082=1049.783,136.077,412.830,171.014,35.194,156.613
C06083=1049.789,136.325,412.810,171.015,35.196,156.613
C06084=1049.796,136.575,412.789,171.018,35.198,156.613
C06085=1049.801,136.823,412.768,171.020,35.200,156.614
C06086=1049.808,137.073,412.747,171.022,35.202,156.614
C06087=1049.814,137.322,412.726,171.024,35.204,156.614
C06088=1049.819,137.570,412.704,171.025,35.206,156.615
C06089=1049.826,137.820,412.683,171.027,35.208,156.615
C06090=1049.832,138.069,412.662,171.029,35.210,156.616
C06091=1049.838,138.318,412.641,171.032,35.212,156.616
C06092=1049.844,138.567,412.619,171.033,35.214,156.616
C06093=1049.850,138.816,412.598,171.035,35.216,156.617
C06094=1049.856,139.065,412.577,171.037,35.218,156.617
C06095=1049.862,139.314,412.556,171.039,35.220,156.617
C06096=1049.868,139.563,412.535,171.041,35.222,156.618
C06097=1049.874,139.812,412.513,171.042,35.224,156.618
C06098=1049.880,140.061,412.492,171.045,35.226,156.618
C06099=1049.886,140.310,412.470,171.047,35.228,156.619
C06100=1049.892,140.559,412.449,171.049,35.230,156.619
C06101=1049.898,140.808,412.428,171.050,35.232,156.620
C06102=1049.905,141.057,412.407,171.052,35.234,156.620
C06103=1049.910,141.306,412.386,171.054,35.237,156.620
C06104=1049.917,141.592,412.360,171.056,35.238,156.621
C06105=1049.924,141.877,412.336,171.059,35.241,156.621
C06106=1049.931,142.162,412.312,171.061,35.243,156.622
C06107=1049.937,142.447,412.287,171.063,35.246,156.622
C06108=1049.944,142.696,412.265,171.065,35.248,156.622
C06109=1049.950,142.946,412.243,171.067,35.250,156.623
C06110=1049.956,143.195,412.222,171.069,35.252,156.623
C06111=1049.961,143.444,412.201,171.071,35.254,156.624
C06112=1049.967,143.693,412.180,171.073,35.256,156.624
C06113=1049.974,143.942,412.158,171.075,35.258,156.624
C06114=1049.979,144.191,412.137,171.077,35.260,156.625
C06115=1049.986,144.440,412.116,171.079,35.262,156.625
C06116=1049.992,144.689,412.094,171.081,35.264,156.625
C06117=1049.999,144.938,412.072,171.082,35.266,156.626
C06118=1050.004,145.186,412.050,171.085,35.268,156.626
C06119=1050.010,145.435,412.029,171.087,35.271,156.627
C06120=1050.017,145.684,412.007,171.089,35.272,156.627
C06121=1050.023,145.934,411.985,171.091,35.274,156.627
C06122=1050.028,146.182,411.964,171.092,35.276,156.628
C06123=1050.034,146.431,411.943,171.094,35.279,156.628
C06124=1050.041,146.681,411.921,171.096,35.281,156.628
C06125=1050.047,146.930,411.899,171.099,35.282,156.629
C06126=1050.053,147.179,411.878,171.101,35.284,156.629
C06127=1050.058,147.428,411.856,171.103,35.286,156.629
C06128=1050.065,147.677,411.835,171.104,35.289,156.630
C06129=1050.071,147.925,411.812,171.106,35.291,156.630
C06130=1050.077,148.175,411.791,171.108,35.293,156.631
C06131=1050.083,148.424,411.769,171.111,35.295,156.631
C06132=1050.088,148.673,411.747,171.113,35.297,156.631
C06133=1050.094,148.922,411.726,171.115,35.299,156.632
C06134=1050.101,149.171,411.704,171.116,35.301,156.632
C06135=1050.107,149.420,411.682,171.118,35.303,156.633
C06136=1050.113,149.669,411.660,171.120,35.305,156.633
C06137=1050.119,149.917,411.639,171.122,35.308,156.633
C06138=1050.125,150.166,411.617,171.125,35.309,156.634
C06139=1050.131,150.415,411.594,171.127,35.311,156.634
C06140=1050.137,150.665,411.572,171.129,35.314,156.635
C06141=1050.143,150.914,411.551,171.130,35.316,156.635
C06142=1050.149,151.162,411.530,171.132,35.318,156.635
C06143=1050.155,151.411,411.507,171.134,35.320,156.636
C06144=1050.160,151.660,411.485,171.137,35.322,156.636
C06145=1050.167,151.910,411.463,171.139,35.324,156.636
C06146=1050.173,152.158,411.441,171.141,35.326,156.637
C06147=1050.179,152.407,411.419,171.142,35.328,156.637
C06148=1050.184,152.656,411.398,171.144,35.330,156.638
C06149=1050.191,152.905,411.375,171.146,35.333,156.638
C06150=1050.197,153.154,411.354,171.148,35.335,156.638
C06151=1050.203,153.403,411.332,171.151,35.336,156.639
C06152=1050.209,153.652,411.310,171.153,35.339,156.639
C06153=1050.215,153.901,411.287,171.155,35.341,156.639
C06154=1050.221,154.150,411.265,171.157,35.343,156.640
C06155=1050.227,154.399,411.243,171.158,35.345,156.640
C06156=1050.233,154.648,411.222,171.160,35.347,156.641
C06157=1050.239,154.896,411.199,171.163,35.350,156.641
C06158=1050.245,155.146,411.177,171.165,35.351,156.641
C06159=1050.251,155.394,411.155,171.167,35.353,156.642
C06160=1050.257,155.644,411.133,171.169,35.356,156.642
C06161=1050.263,155.892,411.111,171.171,35.358,156.643
C06162=1050.269,156.142,411.089,171.173,35.360,156.643
C06163=1050.275,156.390,411.066,171.175,35.362,156.643
C06164=1050.281,156.640,411.044,171.177,35.364,156.644
C06165=1050.288,156.888,411.022,171.179,35.366,156.644
C06166=1050.293,157.137,411.000,171.181,35.368,156.645
C06167=1050.299,157.386,410.978,171.183,35.371,156.645
C06168=1050.306,157.671,410.952,171.185,35.373,156.646
C06169=1050.313,157.956,410.927,171.188,35.375,156.646
C06170=1050.320,158.242,410.901,171.190,35.378,156.646
C06171=1050.326,158.527,410.876,171.193,35.380,156.647
C06172=1050.334,158.835,410.848,171.195,35.383,156.647
C06173=1050.340,159.084,410.826,171.197,35.385,156.648
C06174=1050.346,159.333,410.804,171.199,35.387,156.648
C06175=1050.352,159.582,410.781,171.202,35.390,156.649
C06176=1050.359,159.830,410.759,171.204,35.391,156.649
C06177=1050.364,160.080,410.737,171.206,35.393,156.649
C06178=1050.371,160.328,410.714,171.207,35.396,156.650
C06179=1050.377,160.578,410.693,171.209,35.398,156.650
C06180=1050.382,160.827,410.670,171.211,35.400,156.651
C06181=1050.388,161.075,410.647,171.214,35.402,156.651
C06182=1050.394,161.324,410.624,171.216,35.405,156.651
C06183=1050.400,161.574,410.602,171.218,35.407,156.652
C06184=1050.405,161.822,410.580,171.220,35.409,156.652
C06185=1050.411,162.071,410.557,171.222,35.411,156.653
C06186=1050.417,162.319,410.534,171.225,35.414,156.653
C06187=1050.423,162.569,410.512,171.227,35.416,156.653
C06188=1050.429,162.818,410.489,171.228,35.418,156.654
C06189=1050.434,163.066,410.466,171.230,35.420,156.654
C06190=1050.440,163.315,410.443,171.232,35.423,156.655
C06191=1050.446,163.564,410.421,171.234,35.425,156.655
C06192=1050.452,163.813,410.398,171.237,35.427,156.656
C06193=1050.458,164.062,410.376,171.239,35.429,156.656
C06194=1050.463,164.311,410.353,171.241,35.431,156.656
C06195=1050.469,164.560,410.330,171.243,35.434,156.657
C06196=1050.476,164.809,410.307,171.245,35.436,156.657
C06197=1050.481,165.058,410.284,171.247,35.438,156.658
C06198=1050.487,165.307,410.262,171.250,35.441,156.658
C06199=1050.493,165.555,410.239,171.251,35.443,156.659
C06200=1050.499,165.804,410.216,171.253,35.445,156.659
C06201=1050.505,166.053,410.193,171.255,35.448,156.659
C06202=1050.510,166.302,410.171,171.257,35.449,156.660
C06203=1050.516,166.551,410.148,171.260,35.452,156.660
C06204=1050.522,166.800,410.125,171.262,35.454,156.661
C06205=1050.528,167.049,410.103,171.264,35.456,156.661
C06206=1050.534,167.298,410.080,171.266,35.459,156.661
C06207=1050.540,167.547,410.057,171.268,35.461,156.662
C06208=1050.546,167.796,410.034,171.270,35.463,156.662
C06209=1050.551,168.044,410.011,171.273,35.466,156.663
C06210=1050.558,168.293,409.989,171.275,35.467,156.663
C06211=1050.563,168.542,409.966,171.277,35.470,156.664
C06212=1050.569,168.791,409.943,171.279,35.472,156.664
C06213=1050.576,169.040,409.919,171.281,35.474,156.664
C06214=1050.581,169.289,409.897,171.284,35.477,156.665
C06215=1050.587,169.538,409.874,171.286,35.479,156.665
C06216=1050.593,169.787,409.851,171.288,35.481,156.666
C06217=1050.599,170.035,409.828,171.290,35.484,156.666
C06218=1050.605,170.284,409.805,171.292,35.485,156.667
C06219=1050.611,170.533,409.782,171.294,35.488,156.667
C06220=1050.617,170.782,409.759,171.297,35.490,156.667
C06221=1050.622,171.031,409.736,171.299,35.492,156.668
C06222=1050.629,171.280,409.713,171.301,35.495,156.668
C06223=1050.635,171.529,409.690,171.302,35.497,156.669
C06224=1050.641,171.778,409.667,171.304,35.499,156.669
C06225=1050.647,172.027,409.644,171.307,35.502,156.670
C06226=1050.653,172.275,409.621,171.309,35.503,156.670
C06227=1050.658,172.524,409.598,171.311,35.506,156.670
C06228=1050.666,172.773,409.575,171.313,35.508,156.671
C06229=1050.671,173.022,409.552,171.315,35.510,156.671
C06230=1050.677,173.271,409.529,171.318,35.513,156.672
C06231=1050.683,173.519,409.505,171.320,35.515,156.672
C06232=1050.689,173.789,409.481,171.323,35.517,156.672
C06233=1050.695,174.059,409.455,171.325,35.520,156.673
C06234=1050.703,174.330,409.431,171.327,35.522,156.673
C06235=1050.709,174.599,409.405,171.329,35.525,156.674
C06236=1050.715,174.848,409.382,171.332,35.527,156.674
C06237=1050.721,175.097,409.360,171.334,35.530,156.675
C06238=1050.727,175.346,409.335,171.336,35.531,156.675
C06239=1050.733,175.595,409.313,171.338,35.534,156.676
C06240=1050.739,175.844,409.290,171.340,35.536,156.676
C06241=1050.745,176.092,409.267,171.343,35.538,156.676
C06242=1050.752,176.341,409.243,171.345,35.541,156.677
C06243=1050.758,176.590,409.220,171.347,35.543,156.677
C06244=1050.763,176.839,409.197,171.350,35.545,156.678
C06245=1050.769,177.087,409.174,171.352,35.548,156.678
C06246=1050.776,177.337,409.150,171.355,35.549,156.679
C06247=1050.782,177.585,409.127,171.357,35.552,156.679
C06248=1050.788,177.834,409.104,171.359,35.554,156.680
C06249=1050.794,178.084,409.080,171.361,35.556,156.680
C06250=1050.800,178.332,409.057,171.363,35.559,156.680
C06251=1050.806,178.580,409.034,171.366,35.561,156.681
C06252=1050.813,178.830,409.011,171.368,35.563,156.681
C06253=1050.819,179.078,408.987,171.370,35.566,156.682
C06254=1050.824,179.327,408.964,171.372,35.568,156.682
C06255=1050.831,179.576,408.940,171.374,35.570,156.682
C06256=1050.837,179.825,408.918,171.376,35.572,156.683
C06257=1050.843,180.073,408.894,171.379,35.575,156.683
C06258=1050.849,180.323,408.871,171.381,35.577,156.684
C06259=1050.855,180.571,408.847,171.383,35.579,156.684
C06260=1050.861,180.820,408.824,171.386,35.582,156.685
C06261=1050.868,181.069,408.800,171.388,35.583,156.685
C06262=1050.873,181.318,408.777,171.391,35.586,156.686
C06263=1050.880,181.566,408.754,171.393,35.588,156.686
C06264=1050.886,181.816,408.731,171.395,35.590,156.686
C06265=1050.893,182.064,408.707,171.397,35.593,156.687
C06266=1050.899,182.313,408.684,171.399,35.595,156.687
C06267=1050.905,182.562,408.660,171.402,35.597,156.688
C06268=1050.911,182.811,408.637,171.404,35.600,156.688
C06269=1050.917,183.060,408.613,171.406,35.602,156.689
C06270=1050.923,183.308,408.589,171.409,35.604,156.689
C06271=1050.930,183.557,408.566,171.411,35.606,156.689
C06272=1050.936,183.806,408.542,171.414,35.609,156.690
C06273=1050.942,184.055,408.519,171.416,35.611,156.690
C06274=1050.948,184.304,408.495,171.418,35.613,156.691
C06275=1050.953,184.552,408.471,171.420,35.616,156.691
C06276=1050.960,184.801,408.447,171.422,35.618,156.692
C06277=1050.965,185.050,408.424,171.425,35.621,156.692
C06278=1050.971,185.299,408.400,171.427,35.623,156.693
C06279=1050.977,185.548,408.375,171.429,35.626,156.693
C06280=1050.983,185.796,408.352,171.431,35.628,156.694
C06281=1050.988,186.045,408.327,171.434,35.630,156.694
C06282=1050.995,186.294,408.304,171.437,35.633,156.695
C06283=1051.001,186.543,408.280,171.439,35.635,156.695
C06284=1051.006,186.791,408.256,171.441,35.638,156.695
C06285=1051.013,187.040,408.232,171.443,35.640,156.696
C06286=1051.018,187.289,408.208,171.446,35.643,156.696
C06287=1051.024,187.538,408.184,171.448,35.645,156.697
C06288=1051.029,187.787,408.160,171.450,35.648,156.697
C06289=1051.035,188.035,408.137,171.452,35.650,156.698
C06290=1051.041,188.285,408.112,171.454,35.653,156.698
C06291=1051.047,188.533,408.088,171.458,35.655,156.699
C06292=1051.053,188.782,408.064,171.460,35.658,156.699
C06293=1051.059,189.030,408.040,171.462,35.660,156.700
C06294=1051.065,189.279,408.016,171.464,35.662,156.700
C06295=1051.071,189.528,407.992,171.467,35.665,156.701
C06296=1051.078,189.812,407.965,171.470,35.668,156.701
C06297=1051.085,190.096,407.937,171.472,35.671,156.702
C06298=1051.091,190.381,407.909,171.474,35.674,156.702
C06299=1051.098,190.666,407.882,171.478,35.677,156.703
C06300=1051.104,190.914,407.858,171.480,35.679,156.703
C06301=1051.110,191.163,407.833,171.482,35.682,156.704
C06302=1051.116,191.411,407.809,171.484,35.684,156.704
C06303=1051.122,191.660,407.784,171.486,35.686,156.705
C06304=1051.128,191.908,407.761,171.490,35.689,156.705
C06305=1051.134,192.158,407.736,171.492,35.691,156.706
C06306=1051.140,192.406,407.713,171.494,35.694,156.706
C06307=1051.146,192.655,407.688,171.496,35.696,156.707
C06308=1051.152,192.904,407.664,171.499,35.699,156.707
C06309=1051.158,193.153,407.640,171.501,35.701,156.708
C06310=1051.164,193.401,407.616,171.504,35.704,156.708
C06311=1051.170,193.650,407.591,171.506,35.706,156.709
C06312=1051.176,193.899,407.567,171.508,35.709,156.709
C06313=1051.182,194.148,407.543,171.511,35.711,156.710
C06314=1051.189,194.396,407.518,171.513,35.714,156.710
C06315=1051.194,194.645,407.494,171.515,35.716,156.711
C06316=1051.200,194.894,407.469,171.518,35.718,156.711
C06317=1051.206,195.143,407.446,171.521,35.721,156.712
C06318=1051.212,195.392,407.421,171.523,35.723,156.712
C06319=1051.219,195.640,407.396,171.525,35.726,156.713
C06320=1051.224,195.889,407.372,171.527,35.729,156.713
C06321=1051.231,196.138,407.348,171.531,35.731,156.714
C06322=1051.236,196.386,407.324,171.533,35.734,156.714
C06323=1051.243,196.635,407.300,171.535,35.736,156.715
C06324=1051.249,196.884,407.274,171.537,35.739,156.715
C06325=1051.254,197.133,407.250,171.540,35.741,156.715
C06326=1051.261,197.382,407.226,171.543,35.744,156.716
C06327=1051.267,197.630,407.201,171.545,35.746,156.716
C06328=1051.273,197.878,407.177,171.547,35.749,156.717
C06329=1051.279,198.128,407.153,171.549,35.751,156.717
C06330=1051.286,198.376,407.128,171.553,35.753,156.718
C06331=1051.291,198.625,407.104,171.555,35.757,156.718
C06332=1051.297,198.874,407.079,171.557,35.759,156.719
C06333=1051.304,199.122,407.054,171.559,35.761,156.719
C06334=1051.309,199.371,407.030,171.563,35.764,156.720
C06335=1051.316,199.620,407.006,171.565,35.766,156.720
C06336=1051.322,199.869,406.981,171.567,35.769,156.721
C06337=1051.327,200.117,406.956,171.569,35.771,156.721
C06338=1051.334,200.366,406.932,171.572,35.774,156.722
C06339=1051.340,200.615,406.907,171.575,35.776,156.722
C06340=1051.347,200.864,406.883,171.577,35.779,156.723
C06341=1051.353,201.112,406.858,171.579,35.782,156.723
C06342=1051.358,201.361,406.833,171.582,35.784,156.724
C06343=1051.365,201.609,406.809,171.585,35.787,156.724
C06344=1051.371,201.858,406.784,171.587,35.789,156.725
C06345=1051.377,202.107,406.759,171.589,35.792,156.725
C06346=1051.383,202.356,406.734,171.592,35.795,156.726
C06347=1051.389,202.605,406.709,171.595,35.797,156.726
C06348=1051.394,202.853,406.685,171.597,35.800,156.727
C06349=1051.401,203.102,406.659,171.599,35.802,156.727
C06350=1051.407,203.350,406.635,171.602,35.805,156.728
C06351=1051.413,203.599,406.610,171.605,35.808,156.728
C06352=1051.419,203.848,406.585,171.607,35.810,156.729
C06353=1051.425,204.097,406.561,171.609,35.813,156.729
C06354=1051.431,204.345,406.535,171.612,35.816,156.730
C06355=1051.437,204.593,406.510,171.615,35.818,156.731
C06356=1051.443,204.843,406.486,171.617,35.821,156.731
C06357=1051.449,205.091,406.460,171.620,35.824,156.732
C06358=1051.455,205.340,406.435,171.622,35.826,156.732
C06359=1051.461,205.588,406.410,171.625,35.829,156.733
C06360=1051.486,206.640,406.305,171.849,35.924,156.751
C06361=1051.493,206.888,406.278,171.851,35.927,156.751
C06362=1051.499,207.136,406.252,171.852,35.931,156.752
C06363=1051.506,207.386,406.227,171.855,35.934,156.753
C06364=1051.513,207.634,406.201,171.856,35.938,156.753
C06365=1051.519,207.882,406.175,171.858,35.941,156.754
C06366=1051.526,208.130,406.149,171.861,35.945,156.755
C06367=1051.531,208.378,406.122,171.862,35.948,156.755
C06368=1051.538,208.627,406.097,171.864,35.952,156.756
C06369=1051.544,208.875,406.071,171.867,35.955,156.757
C06370=1051.551,209.124,406.044,171.868,35.959,156.758
C06371=1051.557,209.373,406.018,171.871,35.962,156.758
C06372=1051.563,209.621,405.992,171.872,35.966,156.759
C06373=1051.570,209.870,405.966,171.874,35.969,156.760
C06374=1051.576,210.118,405.939,171.877,35.972,156.760
C06375=1051.582,210.367,405.914,171.878,35.976,156.761
C06376=1051.589,210.615,405.887,171.880,35.980,156.762
C06377=1051.595,210.864,405.861,171.883,35.983,156.763
C06378=1051.602,211.112,405.835,171.884,35.986,156.763
C06379=1051.608,211.361,405.808,171.886,35.990,156.764
C06380=1051.614,211.609,405.782,171.889,35.993,156.765
C06381=1051.621,211.858,405.756,171.890,35.996,156.765
C06382=1051.627,212.107,405.729,171.893,36.000,156.766
C06383=1051.634,212.355,405.703,171.895,36.004,156.767
C06384=1051.639,212.603,405.676,171.896,36.007,156.767
C06385=1051.647,212.852,405.650,171.899,36.011,156.768
C06386=1051.652,213.101,405.624,171.901,36.014,156.769
C06387=1051.659,213.349,405.598,171.902,36.017,156.770
C06388=1051.665,213.598,405.571,171.905,36.021,156.770
C06389=1051.671,213.846,405.545,171.907,36.025,156.771
C06390=1051.678,214.095,405.518,171.908,36.028,156.772
C06391=1051.684,214.343,405.492,171.911,36.031,156.772
C06392=1051.690,214.591,405.465,171.913,36.035,156.773
C06393=1051.696,214.840,405.438,171.915,36.038,156.774
C06394=1051.703,215.088,405.412,171.917,36.041,156.774
C06395=1051.709,215.338,405.385,171.919,36.045,156.775
C06396=1051.716,215.586,405.359,171.921,36.049,156.776
C06397=1051.722,215.835,405.332,171.923,36.052,156.777
C06398=1051.729,216.083,405.306,171.925,36.055,156.777
C06399=1051.735,216.331,405.279,171.927,36.059,156.778
C06400=1051.742,216.580,405.253,171.929,36.062,156.779
C06401=1051.747,216.828,405.226,171.932,36.065,156.779
C06402=1051.754,217.077,405.199,171.934,36.069,156.780
C06403=1051.760,217.325,405.173,171.935,36.073,156.781
C06404=1051.767,217.574,405.146,171.938,36.076,156.781
C06405=1051.773,217.822,405.120,171.940,36.079,156.782
C06406=1051.780,218.071,405.093,171.941,36.083,156.783
C06407=1051.786,218.319,405.066,171.944,36.086,156.784
C06408=1051.793,218.568,405.039,171.946,36.089,156.784
C06409=1051.799,218.816,405.013,171.949,36.093,156.785
C06410=1051.806,219.065,404.986,171.950,36.096,156.786
C06411=1051.811,219.313,404.960,171.952,36.100,156.786
C06412=1051.819,219.562,404.933,171.955,36.103,156.787
C06413=1051.824,219.810,404.907,171.957,36.106,156.788
C06414=1051.831,220.059,404.879,171.958,36.110,156.788
C06415=1051.837,220.307,404.853,171.961,36.113,156.789
C06416=1051.844,220.556,404.826,171.963,36.116,156.790
C06417=1051.850,220.809,404.799,171.965,36.120,156.791
C06418=1051.856,221.063,404.771,171.968,36.123,156.791
C06419=1051.863,221.316,404.743,171.969,36.127,156.792
C06420=1051.870,221.570,404.717,171.972,36.130,156.793
C06421=1051.876,221.818,404.689,171.974,36.134,156.793
C06422=1051.882,222.067,404.662,171.976,36.137,156.794
C06423=1051.888,222.316,404.635,171.978,36.141,156.795
C06424=1051.895,222.563,404.608,171.980,36.144,156.795
C06425=1051.902,222.812,404.581,171.983,36.147,156.796
C06426=1051.907,223.060,404.555,171.985,36.151,156.797
C06427=1051.914,223.309,404.527,171.986,36.154,156.798
C06428=1051.920,223.557,404.500,171.989,36.158,156.798
C06429=1051.926,223.806,404.473,171.991,36.161,156.799
C06430=1051.932,224.054,404.446,171.993,36.164,156.800
C06431=1051.939,224.303,404.419,171.996,36.168,156.800
C06432=1051.946,224.551,404.392,171.997,36.171,156.801
C06433=1051.952,224.800,404.365,172.000,36.174,156.802
C06434=1051.958,225.049,404.338,172.002,36.178,156.803
C06435=1051.964,225.296,404.311,172.004,36.182,156.803
C06436=1051.971,225.545,404.284,172.007,36.185,156.804
C06437=1051.977,225.794,404.256,172.008,36.188,156.805
C06438=1051.983,226.042,404.229,172.010,36.192,156.805
C06439=1051.991,226.290,404.202,172.013,36.195,156.806
C06440=1051.996,226.539,404.176,172.015,36.198,156.807
C06441=1052.003,226.787,404.148,172.018,36.202,156.807
C06442=1052.009,227.036,404.121,172.019,36.205,156.808
C06443=1052.016,227.284,404.094,172.021,36.208,156.809
C06444=1052.022,227.533,404.067,172.024,36.211,156.809
C06445=1052.029,227.782,404.039,172.026,36.215,156.810
C06446=1052.034,228.030,404.012,172.029,36.219,156.811
C06447=1052.041,228.278,403.984,172.031,36.222,156.812
C06448=1052.048,228.526,403.957,172.032,36.225,156.812
C06449=1052.054,228.775,403.931,172.035,36.228,156.813
C06450=1052.061,229.023,403.903,172.037,36.232,156.814
C06451=1052.067,229.272,403.876,172.039,36.235,156.814
C06452=1052.074,229.521,403.848,172.042,36.238,156.815
C06453=1052.080,229.768,403.821,172.044,36.242,156.816
C06454=1052.086,230.018,403.793,172.047,36.245,156.816
C06455=1052.092,230.266,403.765,172.048,36.248,156.817
C06456=1052.098,230.514,403.738,172.050,36.252,156.818
C06457=1052.105,230.762,403.710,172.053,36.256,156.819
C06458=1052.112,231.012,403.683,172.055,36.259,156.819
C06459=1052.118,231.259,403.656,172.058,36.262,156.820
C06460=1052.124,231.508,403.628,172.060,36.266,156.821
C06461=1052.131,231.756,403.601,172.062,36.269,156.821
C06462=1052.137,232.005,403.574,172.064,36.272,156.822
C06463=1052.143,232.253,403.546,172.066,36.275,156.823
C06464=1052.149,232.502,403.518,172.069,36.279,156.823
C06465=1052.156,232.750,403.490,172.071,36.282,156.824
C06466=1052.162,232.998,403.463,172.073,36.285,156.825
C06467=1052.168,233.247,403.436,172.076,36.289,156.826
C06468=1052.174,233.496,403.407,172.078,36.292,156.826
C06469=1052.181,233.743,403.380,172.080,36.295,156.827
C06470=1052.187,233.992,403.352,172.082,36.299,156.828
C06471=1052.194,234.240,403.325,172.084,36.303,156.828
C06472=1052.200,234.489,403.296,172.087,36.306,156.829
C06473=1052.206,234.736,403.270,172.089,36.309,156.830
C06474=1052.212,234.983,403.242,172.092,36.313,156.831
C06475=1052.219,235.230,403.214,172.094,36.316,156.831
C06476=1052.225,235.478,403.186,172.096,36.319,156.832
C06477=1052.231,235.725,403.158,172.099,36.322,156.833
C06478=1052.238,235.972,403.131,172.101,36.326,156.833
C06479=1052.244,236.219,403.104,172.103,36.329,156.834
C06480=1052.250,236.466,403.076,172.105,36.332,156.835
C06481=1052.257,236.714,403.048,172.107,36.336,156.835
C06482=1052.263,236.963,403.020,172.110,36.339,156.836
C06483=1052.270,237.211,402.992,172.112,36.342,156.837
C06484=1052.276,237.459,402.965,172.114,36.346,156.837
C06485=1052.282,237.708,402.937,172.117,36.349,156.838
C06486=1052.288,237.956,402.908,172.119,36.353,156.839
C06487=1052.295,238.205,402.881,172.122,36.356,156.839
C06488=1052.302,238.453,402.853,172.124,36.359,156.840
C06489=1052.308,238.702,402.825,172.126,36.363,156.841
C06490=1052.314,238.949,402.797,172.129,36.366,156.842
C06491=1052.321,239.197,402.769,172.131,36.369,156.842
C06492=1052.327,239.446,402.741,172.134,36.372,156.843
C06493=1052.333,239.695,402.713,172.136,36.376,156.844
C06494=1052.340,239.943,402.685,172.138,36.379,156.844
C06495=1052.346,240.192,402.657,172.141,36.382,156.845
C06496=1052.353,240.440,402.628,172.143,36.386,156.846
C06497=1052.360,240.688,402.601,172.146,36.389,156.846
C06498=1052.366,240.937,402.572,172.148,36.392,156.847
C06499=1052.372,241.185,402.545,172.150,36.396,156.848
C06500=1052.378,241.433,402.517,172.153,36.399,156.849
C06501=1052.385,241.681,402.488,172.155,36.403,156.849
C06502=1052.391,241.930,402.460,172.158,36.405,156.850
C06503=1052.397,242.178,402.432,172.160,36.409,156.851
C06504=1052.403,242.427,402.403,172.162,36.413,156.851
C06505=1052.410,242.675,402.375,172.164,36.416,156.852
C06506=1052.416,242.924,402.347,172.166,36.419,156.853
C06507=1052.423,243.172,402.319,172.169,36.423,156.854
C06508=1052.428,243.420,402.291,172.171,36.426,156.854
C06509=1052.435,243.668,402.263,172.174,36.429,156.855
C06510=1052.441,243.916,402.234,172.176,36.433,156.856
C06511=1052.447,244.165,402.205,172.178,36.436,156.856
C06512=1052.454,244.413,402.177,172.181,36.439,156.857
C06513=1052.460,244.662,402.149,172.183,36.443,156.858
C06514=1052.467,244.910,402.121,172.186,36.446,156.858
C06515=1052.473,245.158,402.092,172.188,36.449,156.859
C06516=1052.479,245.407,402.064,172.191,36.453,156.860
C06517=1052.486,245.655,402.035,172.194,36.456,156.861
C06518=1052.492,245.903,402.007,172.196,36.459,156.861
C06519=1052.498,246.152,401.978,172.199,36.463,156.862
C06520=1052.504,246.400,401.949,172.201,36.466,156.863
C06521=1052.511,246.648,401.921,172.204,36.469,156.863
C06522=1052.517,246.897,401.893,172.206,36.473,156.864
C06523=1052.523,247.145,401.864,172.208,36.476,156.865
C06524=1052.530,247.393,401.835,172.211,36.480,156.866
C06525=1052.535,247.641,401.807,172.213,36.483,156.866
C06526=1052.541,247.889,401.778,172.216,36.487,156.867
C06527=1052.548,248.137,401.749,172.218,36.490,156.868
C06528=1052.554,248.386,401.721,172.221,36.493,156.868
C06529=1052.560,248.630,401.692,172.223,36.497,156.869
C06530=1052.566,248.874,401.664,172.225,36.500,156.870
C06531=1052.573,249.119,401.636,172.228,36.503,156.871
C06532=1052.579,249.363,401.607,172.230,36.507,156.871
C06533=1052.585,249.606,401.579,172.233,36.510,156.872
C06534=1052.591,249.850,401.551,172.235,36.513,156.873
C06535=1052.597,250.095,401.522,172.237,36.516,156.873
C06536=1052.604,250.339,401.494,172.240,36.520,156.874
C06537=1052.610,250.588,401.466,172.242,36.523,156.875
C06538=1052.616,250.836,401.437,172.245,36.526,156.876
C06539=1052.622,251.084,401.408,172.247,36.530,156.876
C06540=1052.628,251.332,401.379,172.250,36.533,156.877
C06541=1052.635,251.581,401.351,172.252,36.536,156.878
C06542=1052.641,251.829,401.322,172.254,36.540,156.878
C06543=1052.648,252.077,401.293,172.258,36.543,156.879
C06544=1052.654,252.325,401.264,172.260,36.546,156.880
C06545=1052.660,252.573,401.235,172.263,36.550,156.881
C06546=1052.667,252.822,401.205,172.265,36.553,156.881
C06547=1052.673,253.071,401.177,172.268,36.556,156.882
C06548=1052.679,253.319,401.148,172.270,36.560,156.883
C06549=1052.685,253.567,401.119,172.272,36.563,156.883
C06550=1052.692,253.815,401.090,172.275,36.566,156.884
C06551=1052.699,254.063,401.061,172.277,36.570,156.885
C06552=1052.705,254.311,401.032,172.281,36.574,156.886
C06553=1052.711,254.559,401.003,172.283,36.576,156.886
C06554=1052.718,254.808,400.974,172.286,36.580,156.887
C06555=1052.724,255.056,400.945,172.288,36.584,156.888
C06556=1052.730,255.304,400.916,172.290,36.586,156.888
C06557=1052.737,255.552,400.887,172.293,36.590,156.889
C06558=1052.743,255.801,400.858,172.295,36.593,156.890
C06559=1052.749,256.049,400.829,172.299,36.597,156.891
C06560=1052.756,256.297,400.799,172.301,36.600,156.891
C06561=1052.762,256.546,400.770,172.304,36.603,156.892
C06562=1052.769,256.794,400.741,172.306,36.607,156.893
C06563=1052.776,257.042,400.713,172.309,36.610,156.893
C06564=1052.782,257.290,400.684,172.311,36.613,156.894
C06565=1052.789,257.539,400.654,172.314,36.617,156.895
C06566=1052.795,257.787,400.625,172.317,36.619,156.895
C06567=1052.801,258.035,400.596,172.319,36.623,156.896
C06568=1052.807,258.283,400.567,172.322,36.627,156.897
C06569=1052.815,258.531,400.537,172.324,36.629,156.898
C06570=1052.821,258.779,400.508,172.327,36.633,156.898
C06571=1052.827,259.027,400.479,172.330,36.637,156.899
C06572=1052.833,259.276,400.450,172.332,36.639,156.900
C06573=1052.840,259.524,400.421,172.335,36.643,156.900
C06574=1052.846,259.773,400.391,172.337,36.646,156.901
C06575=1052.853,260.020,400.362,172.340,36.650,156.902
C06576=1052.860,260.269,400.332,172.343,36.653,156.903
C06577=1052.866,260.517,400.303,172.346,36.656,156.903
C06578=1052.872,260.765,400.274,172.348,36.659,156.904
C06579=1052.879,261.013,400.244,172.350,36.662,156.905
C06580=1052.886,261.261,400.215,172.354,36.666,156.905
C06581=1052.892,261.510,400.186,172.356,36.669,156.906
C06582=1052.899,261.758,400.157,172.359,36.672,156.907
C06583=1052.905,262.006,400.127,172.361,36.676,156.908
C06584=1052.912,262.254,400.098,172.365,36.679,156.908
C06585=1052.918,262.498,400.069,172.367,36.682,156.909
C06586=1052.925,262.740,400.040,172.369,36.685,156.910
C06587=1052.932,262.984,400.011,172.372,36.689,156.910
C06588=1052.937,263.227,399.982,172.374,36.692,156.911
C06589=1052.944,263.470,399.953,172.377,36.695,156.912
C06590=1052.949,263.713,399.924,172.380,36.699,156.913
C06591=1052.956,263.957,399.895,172.383,36.702,156.913
C06592=1052.962,264.200,399.866,172.385,36.705,156.914
C06593=1052.969,264.448,399.836,172.388,36.709,156.915
C06594=1052.974,264.697,399.807,172.391,36.712,156.915
C06595=1052.981,264.944,399.777,172.394,36.715,156.916
C06596=1052.988,265.192,399.747,172.396,36.719,156.917
C06597=1052.994,265.441,399.717,172.398,36.722,156.918
C06598=1053.000,265.688,399.687,172.402,36.725,156.918
C06599=1053.007,265.937,399.658,172.404,36.729,156.919
C06600=1053.013,266.185,399.628,172.407,36.732,156.920
C06601=1053.020,266.434,399.598,172.409,36.736,156.921
C06602=1053.026,266.681,399.568,172.413,36.739,156.921
C06603=1053.032,266.929,399.538,172.415,36.742,156.922
C06604=1053.039,267.178,399.509,172.418,36.746,156.923
C06605=1053.046,267.426,399.479,172.420,36.749,156.923
C06606=1053.052,267.674,399.448,172.424,36.752,156.924
C06607=1053.058,267.922,399.419,172.426,36.756,156.925
C06608=1053.065,268.170,399.389,172.429,36.759,156.926
C06609=1053.071,268.418,399.359,172.432,36.762,156.926
C06610=1053.077,268.666,399.330,172.434,36.766,156.927
C06611=1053.084,268.915,399.299,172.437,36.769,156.928
C06612=1053.090,269.162,399.269,172.439,36.773,156.929
C06613=1053.097,269.411,399.238,172.443,36.776,156.929
C06614=1053.103,269.658,399.209,172.445,36.779,156.930
C06615=1053.109,269.907,399.179,172.448,36.783,156.931
C06616=1053.116,270.155,399.149,172.451,36.786,156.932
C06617=1053.122,270.403,399.119,172.454,36.790,156.932
C06618=1053.129,270.651,399.088,172.456,36.793,156.933
C06619=1053.135,270.899,399.058,172.460,36.796,156.934
C06620=1053.142,271.147,399.028,172.462,36.800,156.934
C06621=1053.147,271.396,398.998,172.465,36.803,156.935
C06622=1053.155,271.644,398.968,172.468,36.807,156.936
C06623=1053.160,271.892,398.938,172.471,36.810,156.937
C06624=1053.168,272.140,398.908,172.473,36.813,156.937
C06625=1053.173,272.388,398.877,172.476,36.817,156.938
C06626=1053.180,272.636,398.847,172.479,36.820,156.939
C06627=1053.186,272.884,398.817,172.481,36.824,156.940
C06628=1053.193,273.132,398.786,172.485,36.826,156.940
C06629=1053.199,273.380,398.756,172.487,36.830,156.941
C06630=1053.206,273.628,398.726,172.490,36.833,156.942
C06631=1053.212,273.876,398.695,172.493,36.837,156.943
C06632=1053.218,274.125,398.665,172.496,36.840,156.943
C06633=1053.225,274.372,398.635,172.499,36.844,156.944
C06634=1053.231,274.621,398.604,172.502,36.847,156.945
C06635=1053.237,274.868,398.574,172.504,36.850,156.946
C06636=1053.244,275.116,398.543,172.508,36.854,156.946
C06637=1053.251,275.365,398.512,172.510,36.857,156.947
C06638=1053.257,275.612,398.482,172.513,36.861,156.948
C06639=1053.263,275.861,398.451,172.516,36.864,156.949
C06640=1053.270,276.108,398.421,172.519,36.868,156.949
C06641=1053.276,276.354,398.391,172.521,36.871,156.950
C06642=1053.282,276.599,398.361,172.525,36.874,156.951
C06643=1053.288,276.845,398.330,172.527,36.878,156.952
C06644=1053.295,277.089,398.300,172.531,36.881,156.952
C06645=1053.301,277.334,398.270,172.533,36.885,156.953
C06646=1053.307,277.580,398.240,172.536,36.888,156.954
C06647=1053.313,277.825,398.209,172.539,36.891,156.955
C06648=1053.321,278.070,398.179,172.542,36.895,156.955
C06649=1053.327,278.319,398.148,172.545,36.898,156.956
C06650=1053.333,278.567,398.118,172.548,36.902,156.957
C06651=1053.340,278.815,398.086,172.550,36.905,156.958
C06652=1053.347,279.063,398.056,172.554,36.909,156.958
C06653=1053.353,279.311,398.026,172.556,36.912,156.959
C06654=1053.359,279.559,397.995,172.560,36.915,156.960
C06655=1053.366,279.807,397.964,172.562,36.919,156.961
C06656=1053.372,280.054,397.933,172.566,36.922,156.961
C06657=1053.378,280.303,397.902,172.568,36.925,156.962
C06658=1053.384,280.551,397.872,172.571,36.929,156.963
C06659=1053.391,280.799,397.840,172.574,36.932,156.964
C06660=1053.397,281.047,397.810,172.577,36.936,156.964
C06661=1053.403,281.294,397.778,172.580,36.939,156.965
C06662=1053.410,281.543,397.748,172.583,36.943,156.966
C06663=1053.416,281.791,397.716,172.586,36.946,156.967
C06664=1053.422,282.039,397.686,172.589,36.950,156.968
C06665=1053.429,282.286,397.655,172.592,36.953,156.968
C06666=1053.436,282.534,397.623,172.595,36.957,156.969
C06667=1053.442,282.783,397.592,172.597,36.960,156.970
C06668=1053.448,283.030,397.561,172.601,36.964,156.971
C06669=1053.455,283.279,397.531,172.603,36.967,156.971
C06670=1053.461,283.527,397.499,172.607,36.971,156.972
C06671=1053.467,283.774,397.468,172.609,36.974,156.973
C06672=1053.474,284.022,397.437,172.613,36.978,156.974
C06673=1053.481,284.270,397.406,172.615,36.981,156.974
C06674=1053.487,284.518,397.375,172.619,36.985,156.975
C06675=1053.493,284.766,397.344,172.621,36.988,156.976
C06676=1053.500,285.014,397.313,172.625,36.992,156.977
C06677=1053.507,285.262,397.281,172.627,36.995,156.978
C06678=1053.513,285.510,397.251,172.631,36.999,156.978
C06679=1053.520,285.758,397.219,172.633,37.002,156.979
C06680=1053.526,286.005,397.188,172.637,37.006,156.980
C06681=1053.533,286.253,397.157,172.639,37.009,156.981
C06682=1053.539,286.501,397.125,172.643,37.013,156.981
C06683=1053.545,286.750,397.094,172.645,37.016,156.982
C06684=1053.552,286.998,397.063,172.649,37.019,156.983
C06685=1053.558,287.246,397.031,172.652,37.023,156.984
C06686=1053.565,287.493,397.000,172.655,37.026,156.985
C06687=1053.571,287.741,396.969,172.658,37.030,156.985
C06688=1053.578,287.989,396.937,172.661,37.033,156.986
C06689=1053.584,288.237,396.906,172.664,37.037,156.987
C06690=1053.591,288.485,396.875,172.667,37.040,156.988
C06691=1053.597,288.733,396.843,172.671,37.044,156.988
C06692=1053.604,288.981,396.812,172.673,37.048,156.989
C06693=1053.610,289.229,396.780,172.677,37.051,156.990
C06694=1053.617,289.476,396.749,172.679,37.055,156.991
C06695=1053.623,289.725,396.717,172.683,37.058,156.992
C06696=1053.629,289.973,396.686,172.686,37.062,156.992
C06697=1053.637,290.227,396.653,172.689,37.065,156.993
C06698=1053.643,290.480,396.621,172.692,37.069,156.994
C06699=1053.649,290.733,396.589,172.695,37.073,156.995
C06700=1053.656,290.988,396.556,172.698,37.076,156.996
C06701=1053.663,291.236,396.524,172.702,37.080,156.997
C06702=1053.669,291.484,396.492,172.704,37.083,156.997
C06703=1053.676,291.731,396.460,172.708,37.087,156.998
C06704=1053.683,291.979,396.429,172.711,37.091,156.999
C06705=1053.688,292.226,396.397,172.714,37.094,157.000
C06706=1053.695,292.474,396.366,172.718,37.097,157.001
C06707=1053.701,292.722,396.334,172.720,37.101,157.001
C06708=1053.707,292.970,396.302,172.724,37.104,157.002
C06709=1053.714,293.218,396.270,172.726,37.108,157.003
C06710=1053.721,293.466,396.239,172.730,37.112,157.004
C06711=1053.727,293.714,396.207,172.733,37.115,157.005
C06712=1053.734,293.962,396.175,172.736,37.119,157.005
C06713=1053.740,294.209,396.143,172.739,37.122,157.006
C06714=1053.747,294.457,396.111,172.743,37.126,157.007
C06715=1053.754,294.705,396.080,172.746,37.130,157.008
C06716=1053.760,294.953,396.047,172.749,37.133,157.009
C06717=1053.767,295.201,396.015,172.752,37.137,157.009
C06718=1053.773,295.449,395.983,172.755,37.140,157.010
C06719=1053.780,295.696,395.951,172.759,37.144,157.011
C06720=1053.786,295.944,395.919,172.761,37.148,157.012
C06721=1053.793,296.192,395.887,172.765,37.151,157.013
C06722=1053.799,296.440,395.855,172.768,37.154,157.013
C06723=1053.805,296.688,395.823,172.771,37.159,157.014
C06724=1053.812,296.935,395.791,172.775,37.162,157.015
C06725=1053.818,297.183,395.758,172.778,37.166,157.016
C06726=1053.824,297.431,395.726,172.781,37.169,157.017
C06727=1053.830,297.679,395.693,172.784,37.173,157.018
C06728=1053.837,297.927,395.662,172.787,37.177,157.019
C06729=1053.843,298.174,395.629,172.791,37.180,157.019
C06730=1053.849,298.422,395.597,172.794,37.184,157.020
C06731=1053.855,298.670,395.564,172.797,37.188,157.021
C06732=1053.862,298.918,395.532,172.800,37.192,157.022
C06733=1053.869,299.166,395.500,172.804,37.195,157.023
C06734=1053.875,299.413,395.468,172.806,37.199,157.023
C06735=1053.882,299.661,395.434,172.810,37.203,157.024
C06736=1053.888,299.910,395.402,172.814,37.206,157.025
C06737=1053.894,300.157,395.370,172.816,37.210,157.026
C06738=1053.901,300.405,395.338,172.820,37.214,157.027
C06739=1053.907,300.652,395.305,172.823,37.218,157.028
C06740=1053.913,300.900,395.273,172.827,37.221,157.029
C06741=1053.920,301.148,395.240,172.830,37.225,157.029
C06742=1053.926,301.396,395.207,172.833,37.229,157.030
C06743=1053.933,301.643,395.175,172.837,37.233,157.031
C06744=1053.939,301.890,395.142,172.839,37.236,157.032
C06745=1053.946,302.139,395.110,172.843,37.239,157.033
C06746=1053.952,302.387,395.077,172.847,37.244,157.034
C06747=1053.958,302.635,395.044,172.850,37.247,157.034
C06748=1053.965,302.882,395.012,172.853,37.251,157.035
C06749=1053.972,303.129,394.980,172.856,37.254,157.036
C06750=1053.978,303.377,394.947,172.860,37.258,157.037
C06751=1053.985,303.625,394.914,172.863,37.262,157.038
C06752=1053.991,303.873,394.881,172.866,37.266,157.039
C06753=1053.998,304.143,394.846,172.870,37.270,157.040
C06754=1054.005,304.412,394.810,172.873,37.274,157.041
C06755=1054.012,304.681,394.775,172.877,37.278,157.042
C06756=1054.020,304.951,394.739,172.881,37.282,157.042
C06757=1054.026,305.199,394.706,172.884,37.286,157.043
C06758=1054.032,305.447,394.673,172.888,37.289,157.044
C06759=1054.039,305.695,394.640,172.892,37.293,157.045
C06760=1054.046,305.942,394.607,172.894,37.297,157.046
C06761=1054.052,306.190,394.575,172.898,37.301,157.047
C06762=1054.059,306.437,394.542,172.901,37.304,157.048
C06763=1054.066,306.686,394.509,172.905,37.308,157.049
C06764=1054.072,306.933,394.477,172.909,37.312,157.049
C06765=1054.078,307.181,394.444,172.911,37.316,157.050
C06766=1054.086,307.428,394.410,172.915,37.320,157.051
C06767=1054.092,307.676,394.377,172.918,37.323,157.052
C06768=1054.098,307.924,394.344,172.922,37.327,157.053
C06769=1054.105,308.172,394.311,172.926,37.330,157.054
C06770=1054.112,308.419,394.279,172.929,37.334,157.055
C06771=1054.119,308.666,394.246,172.932,37.338,157.055
C06772=1054.126,308.914,394.213,172.936,37.342,157.056
C06773=1054.132,309.162,394.180,172.939,37.346,157.057
C06774=1054.139,309.410,394.147,172.943,37.349,157.058
C06775=1054.145,309.657,394.113,172.946,37.353,157.059
C06776=1054.152,309.905,394.081,172.950,37.357,157.060
C06777=1054.159,310.153,394.047,172.953,37.361,157.061
C06778=1054.165,310.400,394.014,172.956,37.365,157.062
C06779=1054.172,310.648,393.981,172.960,37.368,157.062
C06780=1054.178,310.896,393.948,172.964,37.372,157.063
C06781=1054.186,311.144,393.914,172.967,37.376,157.064
C06782=1054.192,311.391,393.882,172.971,37.379,157.065
C06783=1054.199,311.639,393.848,172.974,37.383,157.066
C06784=1054.206,311.886,393.816,172.978,37.387,157.067
C06785=1054.213,312.134,393.782,172.982,37.391,157.068
C06786=1054.220,312.382,393.749,172.984,37.395,157.069
C06787=1054.227,312.630,393.716,172.988,37.398,157.069
C06788=1054.233,312.877,393.682,172.992,37.402,157.070
C06789=1054.240,313.125,393.649,172.995,37.406,157.071
C06790=1054.247,313.372,393.616,172.999,37.410,157.072
C06791=1054.253,313.620,393.582,173.002,37.414,157.073
C06792=1054.259,313.868,393.549,173.006,37.417,157.074
C06793=1054.266,314.116,393.514,173.010,37.421,157.075
C06794=1054.272,314.363,393.481,173.013,37.425,157.076
C06795=1054.279,314.611,393.447,173.016,37.429,157.077
C06796=1054.285,314.858,393.414,173.020,37.433,157.078
C06797=1054.292,315.106,393.379,173.024,37.437,157.079
C06798=1054.298,315.353,393.346,173.027,37.441,157.079
C06799=1054.304,315.602,393.312,173.031,37.445,157.080
C06800=1054.311,315.849,393.279,173.035,37.449,157.081
C06801=1054.317,316.097,393.244,173.038,37.453,157.082
C06802=1054.324,316.344,393.211,173.042,37.457,157.083
C06803=1054.331,316.592,393.176,173.046,37.461,157.084
C06804=1054.337,316.839,393.143,173.048,37.465,157.085
C06805=1054.343,317.087,393.109,173.052,37.469,157.086
C06806=1054.350,317.334,393.076,173.056,37.473,157.087
C06807=1054.356,317.582,393.041,173.059,37.477,157.088
C06808=1054.363,317.829,393.008,173.063,37.481,157.089
C06809=1054.370,318.103,392.970,173.067,37.486,157.090
C06810=1054.378,318.377,392.932,173.072,37.490,157.091
C06811=1054.385,318.651,392.894,173.075,37.495,157.092
C06812=1054.392,318.925,392.857,173.079,37.499,157.093
C06813=1054.398,319.173,392.823,173.083,37.503,157.094
C06814=1054.405,319.420,392.789,173.086,37.507,157.095
C06815=1054.412,319.668,392.755,173.090,37.511,157.096
C06816=1054.418,319.915,392.721,173.094,37.515,157.097
C06817=1054.425,320.163,392.687,173.098,37.519,157.098
C06818=1054.432,320.411,392.653,173.101,37.523,157.099
C06819=1054.438,320.658,392.618,173.105,37.527,157.100
C06820=1054.445,320.905,392.585,173.109,37.531,157.100
C06821=1054.452,321.153,392.550,173.112,37.535,157.101
C06822=1054.458,321.401,392.516,173.116,37.539,157.102
C06823=1054.465,321.648,392.482,173.120,37.543,157.103
C06824=1054.471,321.896,392.448,173.123,37.547,157.104
C06825=1054.479,322.143,392.413,173.127,37.551,157.105
C06826=1054.485,322.391,392.379,173.131,37.555,157.106
C06827=1054.492,322.638,392.346,173.135,37.559,157.107
C06828=1054.498,322.886,392.311,173.138,37.563,157.108
C06829=1054.505,323.134,392.277,173.142,37.568,157.109
C06830=1054.512,323.381,392.242,173.146,37.572,157.110
C06831=1054.519,323.629,392.208,173.149,37.576,157.111
C06832=1054.526,323.876,392.174,173.153,37.579,157.112
C06833=1054.532,324.123,392.139,173.157,37.583,157.113
C06834=1054.539,324.371,392.105,173.161,37.588,157.114
C06835=1054.546,324.619,392.071,173.165,37.592,157.115
C06836=1054.553,324.867,392.036,173.169,37.596,157.116
C06837=1054.560,325.114,392.002,173.173,37.600,157.117
C06838=1054.567,325.362,391.967,173.176,37.604,157.118
C06839=1054.573,325.609,391.933,173.180,37.608,157.119
C06840=1054.580,325.857,391.899,173.184,37.612,157.120
C06841=1054.587,326.104,391.864,173.188,37.617,157.121
C06842=1054.593,326.352,391.829,173.191,37.621,157.122
C06843=1054.600,326.599,391.795,173.195,37.625,157.123
C06844=1054.607,326.847,391.760,173.199,37.628,157.124
C06845=1054.614,327.094,391.726,173.203,37.633,157.125
C06846=1054.621,327.341,391.691,173.207,37.637,157.126
C06847=1054.628,327.589,391.656,173.211,37.641,157.127
C06848=1054.635,327.836,391.622,173.215,37.645,157.128
C06849=1054.642,328.084,391.587,173.219,37.649,157.129
C06850=1054.648,328.332,391.552,173.222,37.653,157.129
C06851=1054.656,328.579,391.518,173.226,37.658,157.131
C06852=1054.662,328.827,391.483,173.230,37.662,157.131
C06853=1054.669,329.074,391.448,173.234,37.666,157.133
C06854=1054.676,329.322,391.414,173.238,37.670,157.134
C06855=1054.683,329.569,391.379,173.242,37.674,157.134
C06856=1054.690,329.817,391.344,173.246,37.678,157.136
C06857=1054.697,330.064,391.309,173.250,37.682,157.136
C06858=1054.704,330.312,391.275,173.253,37.687,157.138
C06859=1054.711,330.559,391.240,173.257,37.691,157.138
C06860=1054.717,330.806,391.205,173.262,37.695,157.140
C06861=1054.723,331.054,391.169,173.266,37.700,157.141
C06862=1054.730,331.301,391.134,173.269,37.704,157.142
C06863=1054.737,331.549,391.099,173.273,37.708,157.143
C06864=1054.744,331.796,391.064,173.277,37.713,157.144
C06865=1054.751,332.065,391.025,173.282,37.717,157.145
C06866=1054.759,332.334,390.987,173.286,37.722,157.146
C06867=1054.766,332.602,390.949,173.291,37.727,157.147
C06868=1054.774,332.871,390.911,173.294,37.731,157.148
C06869=1054.781,333.118,390.876,173.298,37.736,157.149
C06870=1054.787,333.366,390.841,173.302,37.740,157.150
C06871=1054.794,333.613,390.806,173.307,37.744,157.151
C06872=1054.801,333.860,390.770,173.311,37.749,157.152
C06873=1054.808,334.108,390.735,173.314,37.753,157.153
C06874=1054.815,334.355,390.699,173.318,37.757,157.154
C06875=1054.821,334.603,390.663,173.322,37.761,157.155
C06876=1054.828,334.850,390.628,173.327,37.766,157.157
C06877=1054.835,335.098,390.593,173.331,37.770,157.158
C06878=1054.842,335.345,390.558,173.334,37.774,157.159
C06879=1054.848,335.592,390.523,173.338,37.779,157.160
C06880=1054.856,335.840,390.487,173.343,37.783,157.161
C06881=1054.863,336.087,390.451,173.347,37.788,157.162
C06882=1054.870,336.334,390.416,173.351,37.792,157.163
C06883=1054.876,336.582,390.381,173.355,37.797,157.164
C06884=1054.883,336.830,390.344,173.359,37.801,157.165
C06885=1054.890,337.077,390.309,173.363,37.806,157.166
C06886=1054.897,337.324,390.273,173.367,37.810,157.167
C06887=1054.903,337.571,390.238,173.371,37.815,157.168
C06888=1054.910,337.819,390.203,173.376,37.819,157.169
C06889=1054.918,338.066,390.166,173.380,37.823,157.170
C06890=1054.924,338.314,390.131,173.383,37.828,157.172
C06891=1054.931,338.561,390.095,173.387,37.832,157.173
C06892=1054.937,338.808,390.060,173.392,37.837,157.174
C06893=1054.944,339.056,390.023,173.396,37.841,157.175
C06894=1054.951,339.303,389.988,173.400,37.846,157.176
C06895=1054.958,339.550,389.952,173.405,37.850,157.177
C06896=1054.965,339.798,389.916,173.409,37.855,157.178
C06897=1054.972,340.045,389.880,173.412,37.859,157.179
C06898=1054.979,340.292,389.844,173.417,37.864,157.180
C06899=1054.986,340.540,389.808,173.421,37.868,157.181
C06900=1054.993,340.787,389.772,173.425,37.873,157.183
C06901=1055.000,341.034,389.736,173.430,37.878,157.184
C06902=1055.006,341.282,389.700,173.434,37.882,157.185
C06903=1055.014,341.529,389.664,173.438,37.886,157.186
C06904=1055.020,341.776,389.627,173.442,37.891,157.187
C06905=1055.027,342.024,389.592,173.446,37.895,157.188
C06906=1055.034,342.271,389.556,173.450,37.900,157.189
C06907=1055.041,342.518,389.520,173.455,37.905,157.190
C06908=1055.048,342.765,389.484,173.459,37.909,157.191
C06909=1055.055,343.013,389.447,173.463,37.914,157.193
C06910=1055.062,343.260,389.412,173.468,37.919,157.194
C06911=1055.069,343.508,389.375,173.472,37.923,157.195
C06912=1055.076,343.755,389.339,173.476,37.928,157.196
C06913=1055.082,344.002,389.303,173.480,37.933,157.197
C06914=1055.090,344.249,389.267,173.484,37.937,157.198
C06915=1055.096,344.496,389.230,173.489,37.942,157.199
C06916=1055.103,344.744,389.193,173.493,37.946,157.201
C06917=1055.110,344.991,389.157,173.498,37.951,157.202
C06918=1055.117,345.238,389.121,173.502,37.956,157.203
C06919=1055.124,345.485,389.085,173.506,37.960,157.204
C06920=1055.131,345.733,389.048,173.511,37.965,157.205
C06921=1055.139,345.997,389.009,173.515,37.970,157.206
C06922=1055.146,346.262,388.969,173.520,37.975,157.208
C06923=1055.153,346.526,388.931,173.525,37.980,157.209
C06924=1055.161,346.790,388.891,173.529,37.985,157.210
C06925=1055.168,347.037,388.855,173.534,37.990,157.211
C06926=1055.175,347.285,388.818,173.538,37.995,157.213
C06927=1055.182,347.532,388.782,173.543,38.000,157.214
C06928=1055.189,347.780,388.745,173.547,38.005,157.215
C06929=1055.196,348.027,388.708,173.552,38.010,157.216
C06930=1055.203,348.273,388.672,173.555,38.014,157.217
C06931=1055.210,348.521,388.635,173.560,38.019,157.218
C06932=1055.216,348.768,388.598,173.564,38.024,157.220
C06933=1055.224,349.015,388.562,173.569,38.028,157.221
C06934=1055.231,349.263,388.525,173.573,38.033,157.222
C06935=1055.238,349.509,388.488,173.578,38.038,157.223
C06936=1055.245,349.757,388.451,173.582,38.043,157.224
C06937=1055.253,350.004,388.414,173.587,38.048,157.226
C06938=1055.259,350.251,388.377,173.591,38.053,157.227
C06939=1055.266,350.498,388.340,173.596,38.058,157.228
C06940=1055.273,350.746,388.303,173.600,38.063,157.229
C06941=1055.281,350.993,388.266,173.605,38.067,157.230
C06942=1055.287,351.240,388.230,173.609,38.072,157.232
C06943=1055.295,351.487,388.192,173.614,38.077,157.233
C06944=1055.302,351.735,388.155,173.618,38.082,157.234
C06945=1055.308,351.981,388.118,173.623,38.087,157.235
C06946=1055.316,352.228,388.081,173.627,38.092,157.237
C06947=1055.322,352.476,388.044,173.632,38.097,157.238
C06948=1055.330,352.723,388.006,173.636,38.102,157.239
C06949=1055.336,352.969,387.969,173.641,38.107,157.240
C06950=1055.343,353.217,387.932,173.645,38.112,157.242
C06951=1055.351,353.464,387.895,173.650,38.117,157.243
C06952=1055.358,353.712,387.857,173.655,38.122,157.244
C06953=1055.364,353.958,387.820,173.659,38.127,157.245
C06954=1055.372,354.205,387.783,173.664,38.132,157.246
C06955=1055.379,354.452,387.745,173.668,38.137,157.248
C06956=1055.386,354.700,387.708,173.673,38.142,157.249
C06957=1055.393,354.947,387.671,173.677,38.147,157.250
C06958=1055.400,355.194,387.634,173.682,38.152,157.252
C06959=1055.407,355.441,387.596,173.687,38.157,157.253
C06960=1055.414,355.688,387.559,173.691,38.162,157.254
C06961=1055.421,355.935,387.521,173.696,38.167,157.255
C06962=1055.429,356.182,387.484,173.701,38.172,157.257
C06963=1055.436,356.429,387.446,173.705,38.177,157.258
C06964=1055.443,356.676,387.408,173.710,38.182,157.259
C06965=1055.450,356.924,387.371,173.715,38.188,157.261
C06966=1055.458,357.171,387.333,173.720,38.193,157.262
C06967=1055.465,357.418,387.296,173.725,38.198,157.263
C06968=1055.473,357.664,387.258,173.729,38.203,157.264
C06969=1055.480,357.911,387.220,173.734,38.208,157.266
C06970=1055.486,358.158,387.182,173.739,38.213,157.267
C06971=1055.493,358.405,387.145,173.743,38.218,157.268
C06972=1055.500,358.652,387.107,173.748,38.223,157.270
C06973=1055.508,358.899,387.069,173.753,38.229,157.271
C06974=1055.515,359.146,387.032,173.757,38.234,157.272
C06975=1055.521,359.394,386.993,173.762,38.239,157.274
C06976=1055.529,359.640,386.955,173.767,38.245,157.275
C06977=1055.537,359.910,386.914,173.773,38.250,157.276
C06978=1055.544,360.179,386.872,173.778,38.256,157.278
C06979=1055.553,360.448,386.831,173.783,38.262,157.279
C06980=1055.561,360.718,386.790,173.788,38.267,157.281
C06981=1055.568,360.965,386.752,173.793,38.273,157.282
C06982=1055.575,361.212,386.713,173.797,38.278,157.283
C06983=1055.582,361.459,386.676,173.802,38.283,157.285
C06984=1055.590,361.705,386.638,173.808,38.289,157.286
C06985=1055.596,361.953,386.599,173.813,38.294,157.287
C06986=1055.604,362.199,386.561,173.817,38.300,157.289
C06987=1055.611,362.446,386.524,173.822,38.304,157.290
C06988=1055.619,362.694,386.484,173.827,38.310,157.291
C06989=1055.626,362.941,386.446,173.832,38.315,157.293
C06990=1055.633,363.188,386.409,173.836,38.321,157.294
C06991=1055.640,363.434,386.370,173.842,38.326,157.296
C06992=1055.648,363.681,386.332,173.847,38.332,157.297
C06993=1055.654,363.928,386.293,173.852,38.337,157.298
C06994=1055.662,364.176,386.255,173.857,38.343,157.300
C06995=1055.669,364.422,386.216,173.861,38.348,157.301
C06996=1055.677,364.669,386.178,173.867,38.354,157.303
C06997=1055.684,364.916,386.139,173.872,38.359,157.304
C06998=1055.691,365.162,386.101,173.877,38.364,157.305
C06999=1055.698,365.409,386.062,173.882,38.370,157.307
C07000=1055.705,365.657,386.023,173.886,38.375,157.308
C07001=1055.713,365.904,385.985,173.891,38.381,157.310
C07002=1055.719,366.151,385.946,173.897,38.386,157.311
C07003=1055.727,366.397,385.908,173.902,38.392,157.313
C07004=1055.734,366.645,385.869,173.907,38.398,157.314
C07005=1055.742,366.891,385.830,173.912,38.403,157.315
C07006=1055.749,367.137,385.791,173.916,38.409,157.317
C07007=1055.756,367.384,385.752,173.922,38.415,157.318
C07008=1055.764,367.631,385.714,173.927,38.420,157.320
C07009=1055.771,367.878,385.675,173.932,38.425,157.321
C07010=1055.778,368.125,385.637,173.937,38.431,157.322
C07011=1055.786,368.372,385.597,173.943,38.437,157.324
C07012=1055.793,368.619,385.558,173.948,38.442,157.325
C07013=1055.801,368.865,385.520,173.953,38.448,157.327
C07014=1055.808,369.113,385.480,173.958,38.454,157.328
C07015=1055.815,369.359,385.442,173.962,38.459,157.330
C07016=1055.823,369.606,385.402,173.968,38.465,157.331
C07017=1055.830,369.853,385.363,173.973,38.471,157.333
C07018=1055.838,370.099,385.325,173.978,38.477,157.334
C07019=1055.845,370.346,385.285,173.984,38.482,157.336
C07020=1055.852,370.593,385.246,173.989,38.488,157.337
C07021=1055.861,370.840,385.207,173.994,38.494,157.339
C07022=1055.867,371.086,385.168,173.999,38.499,157.340
C07023=1055.875,371.334,385.129,174.005,38.505,157.342
C07024=1055.883,371.580,385.090,174.010,38.511,157.343
C07025=1055.890,371.827,385.051,174.015,38.517,157.345
C07026=1055.897,372.074,385.011,174.021,38.523,157.346
C07027=1055.905,372.321,384.971,174.026,38.529,157.348
C07028=1055.912,372.567,384.933,174.031,38.534,157.349
C07029=1055.920,372.814,384.893,174.036,38.540,157.351
C07030=1055.927,373.060,384.854,174.042,38.546,157.352
C07031=1055.935,373.308,384.814,174.047,38.552,157.354
C07032=1055.942,373.554,384.775,174.052,38.558,157.355
C07033=1055.954,373.957,384.709,174.061,38.568,157.358
C07034=1055.966,374.359,384.646,174.070,38.577,157.360
C07035=1055.978,374.762,384.581,174.078,38.587,157.363
C07036=1055.990,375.164,384.516,174.087,38.597,157.365
C07037=1055.998,375.411,384.476,174.093,38.603,157.367
C07038=1056.005,375.658,384.436,174.098,38.609,157.369
C07039=1056.013,375.904,384.396,174.103,38.615,157.370
C07040=1056.020,376.151,384.356,174.109,38.621,157.372
C07041=1056.028,376.398,384.316,174.114,38.627,157.373
C07042=1056.036,376.644,384.277,174.120,38.633,157.375
C07043=1056.044,376.891,384.237,174.126,38.639,157.376
C07044=1056.051,377.138,384.197,174.131,38.645,157.378
C07045=1056.058,377.384,384.158,174.137,38.651,157.380
C07046=1056.066,377.631,384.118,174.142,38.657,157.381
C07047=1056.073,377.877,384.077,174.148,38.664,157.383
C07048=1056.081,378.124,384.037,174.153,38.670,157.385
C07049=1056.088,378.370,383.997,174.158,38.676,157.386
C07050=1056.096,378.617,383.957,174.164,38.682,157.388
C07051=1056.104,378.864,383.917,174.170,38.688,157.389
C07052=1056.112,379.110,383.877,174.176,38.694,157.391
C07053=1056.119,379.357,383.837,174.181,38.700,157.393
C07054=1056.127,379.603,383.797,174.187,38.707,157.394
C07055=1056.135,379.850,383.757,174.192,38.713,157.396
C07056=1056.142,380.097,383.717,174.197,38.719,157.398
C07057=1056.150,380.343,383.676,174.204,38.726,157.399
C07058=1056.158,380.590,383.636,174.209,38.731,157.401
C07059=1056.166,380.836,383.596,174.215,38.738,157.403
C07060=1056.173,381.083,383.555,174.220,38.744,157.404
C07061=1056.185,381.462,383.493,174.230,38.754,157.407
C07062=1056.196,381.840,383.430,174.238,38.764,157.410
C07063=1056.208,382.218,383.368,174.247,38.774,157.412
C07064=1056.220,382.597,383.306,174.256,38.784,157.415
C07065=1056.228,382.844,383.265,174.261,38.790,157.416
C07066=1056.236,383.090,383.224,174.268,38.797,157.418
C07067=1056.243,383.337,383.184,174.273,38.803,157.420
C07068=1056.251,383.583,383.143,174.279,38.810,157.422
C07069=1056.259,383.830,383.102,174.284,38.816,157.423
C07070=1056.266,384.076,383.061,174.291,38.823,157.425
C07071=1056.274,384.323,383.021,174.297,38.829,157.427
C07072=1056.281,384.569,382.979,174.302,38.836,157.428
C07073=1056.289,384.815,382.939,174.309,38.843,157.430
C07074=1056.297,385.062,382.898,174.314,38.849,157.432
C07075=1056.305,385.308,382.857,174.320,38.855,157.434
C07076=1056.313,385.555,382.816,174.326,38.862,157.436
C07077=1056.320,385.801,382.775,174.332,38.869,157.437
C07078=1056.328,386.047,382.734,174.338,38.875,157.439
C07079=1056.336,386.294,382.694,174.344,38.882,157.441
C07080=1056.344,386.541,382.652,174.350,38.888,157.443
C07081=1056.352,386.787,382.611,174.355,38.895,157.444
C07082=1056.360,387.033,382.570,174.362,38.902,157.446
C07083=1056.368,387.280,382.529,174.368,38.909,157.448
C07084=1056.375,387.526,382.488,174.374,38.915,157.450
C07085=1056.385,387.845,382.434,174.382,38.924,157.452
C07086=1056.396,388.165,382.381,174.390,38.933,157.455
C07087=1056.406,388.485,382.327,174.398,38.942,157.457
C07088=1056.417,388.805,382.273,174.405,38.950,157.459
C07089=1056.425,389.051,382.232,174.412,38.957,157.461
C07090=1056.433,389.297,382.191,174.417,38.964,157.463
C07091=1056.441,389.544,382.149,174.424,38.971,157.465
C07092=1056.449,389.790,382.108,174.430,38.978,157.467
C07093=1056.456,390.037,382.067,174.436,38.984,157.468
C07094=1056.465,390.283,382.025,174.442,38.992,157.470
C07095=1056.473,390.529,381.983,174.449,38.999,157.472
C07096=1056.480,390.776,381.942,174.455,39.006,157.474
C07097=1056.488,391.022,381.899,174.461,39.013,157.476
C07098=1056.497,391.268,381.858,174.467,39.020,157.478
C07099=1056.504,391.514,381.816,174.474,39.026,157.480
C07100=1056.512,391.761,381.775,174.479,39.033,157.482
C07101=1056.521,392.007,381.733,174.486,39.041,157.484
C07102=1056.529,392.254,381.691,174.492,39.048,157.486
C07103=1056.536,392.499,381.649,174.499,39.055,157.487
C07104=1056.544,392.745,381.607,174.505,39.062,157.490
C07105=1056.553,392.992,381.565,174.511,39.069,157.491
C07106=1056.560,393.238,381.523,174.518,39.076,157.493
C07107=1056.569,393.484,381.481,174.524,39.083,157.495
C07108=1056.576,393.730,381.439,174.531,39.091,157.497
C07109=1056.584,393.977,381.397,174.537,39.098,157.499
C07110=1056.592,394.223,381.355,174.544,39.105,157.501
C07111=1056.601,394.469,381.312,174.550,39.112,157.503
C07112=1056.609,394.715,381.270,174.556,39.119,157.505
C07113=1056.617,394.961,381.228,174.563,39.127,157.507
C07114=1056.625,395.207,381.186,174.569,39.134,157.509
C07115=1056.633,395.454,381.144,174.576,39.141,157.511
C07116=1056.641,395.700,381.101,174.583,39.148,157.513
C07117=1056.649,395.946,381.059,174.588,39.156,157.515
C07118=1056.657,396.193,381.017,174.595,39.163,157.517
C07119=1056.666,396.439,380.974,174.602,39.171,157.519
C07120=1056.673,396.685,380.932,174.608,39.178,157.521
C07121=1056.682,396.931,380.889,174.615,39.185,157.523
C07122=1056.690,397.178,380.846,174.622,39.193,157.525
C07123=1056.698,397.423,380.804,174.628,39.200,157.527
C07124=1056.706,397.670,380.761,174.635,39.208,157.529
C07125=1056.714,397.916,380.718,174.642,39.215,157.532
C07126=1056.723,398.162,380.676,174.649,39.223,157.534
C07127=1056.731,398.408,380.633,174.655,39.230,157.536
C07128=1056.739,398.654,380.590,174.662,39.238,157.538
C07129=1056.747,398.900,380.548,174.669,39.246,157.540
C07130=1056.755,399.147,380.504,174.676,39.253,157.542
C07131=1056.764,399.393,380.461,174.682,39.261,157.544
C07132=1056.772,399.639,380.418,174.689,39.268,157.546
C07133=1056.780,399.884,380.376,174.696,39.276,157.548
C07134=1056.788,400.131,380.333,174.703,39.283,157.550
C07135=1056.797,400.377,380.290,174.709,39.291,157.553
C07136=1056.805,400.623,380.247,174.716,39.299,157.555
C07137=1056.813,400.869,380.204,174.723,39.307,157.557
C07138=1056.821,401.115,380.161,174.730,39.315,157.559
C07139=1056.830,401.362,380.118,174.737,39.322,157.561
C07140=1056.838,401.608,380.075,174.744,39.330,157.563
C07141=1056.850,401.945,380.016,174.753,39.341,157.566
C07142=1056.861,402.282,379.956,174.763,39.351,157.569
C07143=1056.873,402.619,379.897,174.773,39.362,157.572
C07144=1056.885,402.956,379.837,174.781,39.373,157.575
C07145=1056.893,403.203,379.793,174.789,39.381,157.578
C07146=1056.901,403.449,379.750,174.796,39.389,157.580
C07147=1056.909,403.695,379.707,174.803,39.397,157.582
C07148=1056.918,403.941,379.663,174.810,39.405,157.584
C07149=1056.926,404.187,379.620,174.817,39.413,157.587
C07150=1056.934,404.432,379.575,174.824,39.421,157.589
C07151=1056.943,404.678,379.532,174.831,39.429,157.591
C07152=1056.951,404.925,379.488,174.839,39.437,157.593
C07153=1056.960,405.171,379.445,174.846,39.445,157.595
C07154=1056.968,405.417,379.400,174.853,39.453,157.598
C07155=1056.976,405.663,379.357,174.860,39.461,157.600
C07156=1056.985,405.909,379.313,174.868,39.470,157.602
C07157=1056.994,406.155,379.269,174.875,39.478,157.605
C07158=1057.002,406.401,379.225,174.882,39.486,157.607
C07159=1057.010,406.647,379.181,174.889,39.494,157.609
C07160=1057.019,406.893,379.137,174.897,39.503,157.612
C07161=1057.027,407.139,379.092,174.904,39.511,157.614
C07162=1057.036,407.384,379.049,174.911,39.519,157.616
C07163=1057.044,407.630,379.004,174.919,39.528,157.619
C07164=1057.053,407.876,378.960,174.927,39.536,157.621
C07165=1057.061,408.122,378.917,174.934,39.544,157.624
C07166=1057.070,408.369,378.872,174.941,39.553,157.626
C07167=1057.078,408.614,378.827,174.949,39.561,157.628
C07168=1057.087,408.859,378.783,174.956,39.570,157.631
C07169=1057.096,409.106,378.738,174.964,39.578,157.633
C07170=1057.104,409.351,378.694,174.971,39.586,157.635
C07171=1057.113,409.598,378.650,174.979,39.595,157.638
C07172=1057.121,409.843,378.606,174.987,39.604,157.640
C07173=1057.130,410.090,378.561,174.994,39.612,157.643
C07174=1057.139,410.335,378.516,175.002,39.621,157.645
C07175=1057.148,410.581,378.472,175.010,39.630,157.648
C07176=1057.157,410.828,378.427,175.017,39.638,157.650
C07177=1057.166,411.072,378.383,175.025,39.647,157.653
C07178=1057.174,411.319,378.338,175.032,39.656,157.655
C07179=1057.182,411.565,378.294,175.041,39.664,157.658
C07180=1057.192,411.810,378.249,175.048,39.673,157.660
C07181=1057.201,412.056,378.204,175.056,39.681,157.663
C07182=1057.209,412.302,378.159,175.064,39.690,157.665
C07183=1057.218,412.548,378.114,175.072,39.699,157.668
C07184=1057.228,412.794,378.069,175.079,39.708,157.670
C07185=1057.237,413.039,378.024,175.088,39.717,157.673
C07186=1057.245,413.286,377.979,175.095,39.725,157.675
C07187=1057.254,413.531,377.934,175.103,39.734,157.678
C07188=1057.263,413.776,377.889,175.111,39.743,157.680
C07189=1057.272,414.022,377.844,175.119,39.752,157.683
C07190=1057.281,414.269,377.799,175.128,39.761,157.686
C07191=1057.290,414.515,377.754,175.135,39.770,157.688
C07192=1057.298,414.760,377.709,175.144,39.779,157.691
C07193=1057.307,415.006,377.663,175.152,39.789,157.694
C07194=1057.315,415.252,377.617,175.160,39.797,157.696
C07195=1057.324,415.497,377.572,175.168,39.807,157.699
C07196=1057.333,415.743,377.527,175.175,39.816,157.701
C07197=1057.346,416.086,377.462,175.187,39.828,157.705
C07198=1057.359,416.429,377.399,175.199,39.841,157.709
C07199=1057.372,416.772,377.336,175.211,39.854,157.713
C07200=1057.384,417.115,377.272,175.222,39.867,157.716
C07201=1057.393,417.361,377.227,175.230,39.877,157.719
C07202=1057.402,417.606,377.181,175.239,39.886,157.722
C07203=1057.411,417.852,377.135,175.247,39.895,157.725
C07204=1057.420,418.097,377.088,175.256,39.904,157.727
C07205=1057.429,418.343,377.043,175.264,39.914,157.730
C07206=1057.438,418.588,376.997,175.272,39.923,157.733
C07207=1057.447,418.834,376.951,175.281,39.933,157.736
C07208=1057.456,419.079,376.905,175.290,39.942,157.738
C07209=1057.466,419.326,376.860,175.298,39.952,157.741
C07210=1057.475,419.571,376.813,175.307,39.961,157.744
C07211=1057.485,419.816,376.767,175.315,39.970,157.747
C07212=1057.493,420.062,376.721,175.324,39.980,157.750
C07213=1057.502,420.308,376.675,175.332,39.990,157.752
C07214=1057.512,420.554,376.629,175.341,40.000,157.755
C07215=1057.521,420.799,376.582,175.350,40.009,157.758
C07216=1057.530,421.044,376.536,175.359,40.019,157.761
C07217=1057.539,421.289,376.490,175.367,40.029,157.764
C07218=1057.548,421.536,376.442,175.376,40.039,157.767
C07219=1057.558,421.781,376.396,175.385,40.048,157.770
C07220=1057.566,422.026,376.349,175.394,40.058,157.773
C07221=1057.576,422.272,376.302,175.403,40.068,157.776
C07222=1057.586,422.517,376.256,175.412,40.078,157.779
C07223=1057.594,422.762,376.210,175.421,40.088,157.782
C07224=1057.604,423.008,376.163,175.430,40.098,157.784
C07225=1057.614,423.253,376.116,175.439,40.108,157.787
C07226=1057.623,423.499,376.069,175.448,40.118,157.790
C07227=1057.632,423.744,376.022,175.456,40.128,157.793
C07228=1057.641,423.990,375.975,175.466,40.138,157.796
C07229=1057.651,424.235,375.929,175.475,40.148,157.800
C07230=1057.660,424.481,375.881,175.485,40.158,157.803
C07231=1057.670,424.725,375.834,175.494,40.168,157.805
C07232=1057.680,424.971,375.788,175.503,40.178,157.809
C07233=1057.689,425.216,375.740,175.513,40.189,157.812
C07234=1057.699,425.461,375.693,175.522,40.199,157.815
C07235=1057.708,425.708,375.646,175.531,40.209,157.818
C07236=1057.717,425.952,375.599,175.540,40.219,157.821
C07237=1057.727,426.198,375.551,175.549,40.229,157.824
C07238=1057.737,426.443,375.504,175.559,40.240,157.827
C07239=1057.746,426.688,375.457,175.568,40.250,157.830
C07240=1057.755,426.934,375.409,175.578,40.261,157.833
C07241=1057.766,427.179,375.362,175.588,40.271,157.837
C07242=1057.774,427.424,375.314,175.597,40.282,157.840
C07243=1057.784,427.669,375.267,175.606,40.292,157.843
C07244=1057.794,427.915,375.219,175.616,40.303,157.846
C07245=1057.804,428.160,375.171,175.626,40.313,157.849
C07246=1057.813,428.405,375.123,175.635,40.324,157.853
C07247=1057.823,428.650,375.076,175.645,40.335,157.856
C07248=1057.832,428.895,375.028,175.655,40.345,157.859
C07249=1057.842,429.140,374.980,175.665,40.356,157.862
C07250=1057.852,429.386,374.933,175.674,40.367,157.866
C07251=1057.862,429.631,374.884,175.685,40.377,157.869
C07252=1057.872,429.876,374.836,175.694,40.389,157.872
C07253=1057.886,430.240,374.765,175.709,40.404,157.877
C07254=1057.901,430.605,374.693,175.724,40.421,157.882
C07255=1057.915,430.970,374.621,175.739,40.437,157.887
C07256=1057.929,431.334,374.550,175.754,40.453,157.892
C07257=1057.940,431.579,374.501,175.764,40.464,157.896
C07258=1057.949,431.824,374.452,175.774,40.476,157.899
C07259=1057.959,432.069,374.404,175.785,40.487,157.902
C07260=1057.969,432.314,374.355,175.794,40.498,157.906
C07261=1057.979,432.559,374.307,175.805,40.509,157.909
C07262=1057.988,432.804,374.258,175.816,40.520,157.913
C07263=1057.998,433.049,374.209,175.825,40.531,157.916
C07264=1058.008,433.294,374.161,175.836,40.543,157.920
C07265=1058.019,433.539,374.112,175.847,40.554,157.923
C07266=1058.028,433.784,374.063,175.857,40.565,157.927
C07267=1058.038,434.029,374.014,175.868,40.577,157.930
C07268=1058.049,434.274,373.965,175.879,40.588,157.934
C07269=1058.059,434.519,373.916,175.888,40.600,157.937
C07270=1058.069,434.764,373.867,175.899,40.611,157.941
C07271=1058.079,435.009,373.818,175.910,40.623,157.945
C07272=1058.089,435.254,373.769,175.921,40.634,157.948
C07273=1058.099,435.498,373.720,175.932,40.645,157.952
C07274=1058.109,435.744,373.671,175.942,40.657,157.955
C07275=1058.119,435.988,373.622,175.953,40.669,157.959
C07276=1058.130,436.233,373.572,175.964,40.680,157.963
C07277=1058.140,436.477,373.523,175.975,40.692,157.966
C07278=1058.151,436.722,373.473,175.986,40.704,157.970
C07279=1058.161,436.968,373.424,175.997,40.716,157.974
